KUKA KRL program: MyProgram_107().src

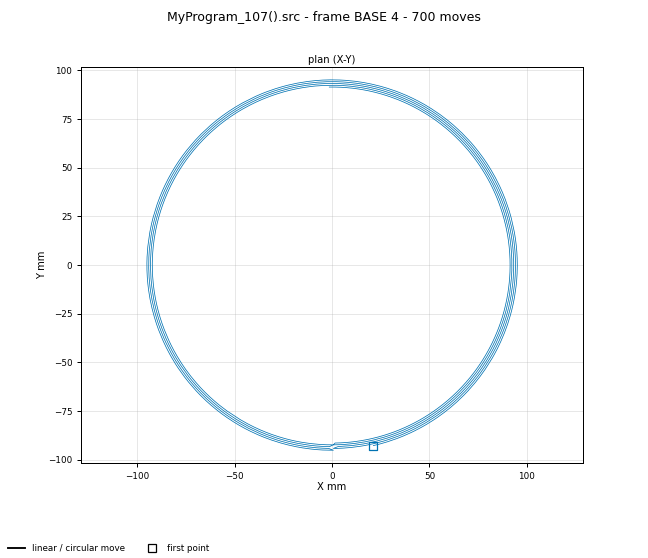
[picture p0: tool path of MyProgram_107().src in frame BASE 4, 700 of 700 moves have a stored position in this frame; points joined in program order, loops and branches not executed]
&ACCESS RVP
&REL 1
&PARAM TEMPLATE = C:\KRC\Roboter\Template\vorgabe
&PARAM EDITMASK = *
DEF MyProgram_107()
; ---- Setting reference (Base) ----
$BASE = BASE_DATA[4]

; --------------------------
; ---- Setting tool (TCP) ----
$TOOL = TOOL_DATA[3]
; --------------------------

$VEL.CP = VEL_APROX_PRINT
Startdeposition()
$VEL.CP = VEL_PRINT
LIN {X 21.2015,Y -92.7621,Z 95,A -81.1872,B 24.9355,C -1.8549,E1 25.0369,E2 526.4414} C_DIS
LIN {X 24.5046,Y -91.9451,Z 95,A -78.7968,B 24.9345,C -1.8695,E1 25.0434,E2 524.0201} C_DIS
LIN {X 28.303,Y -90.8473,Z 95,A -76.2009,B 24.9337,C -1.8802,E1 25.0504,E2 521.4036} C_DIS
LIN {X 33.1897,Y -89.179,Z 95,A -73.7268,B 24.9351,C -1.8608,E1 25.0568,E2 518.9806} C_DIS
LIN {X 36.3029,Y -87.9579,Z 95,A -71.0756,B 24.9332,C -1.8872,E1 25.0638,E2 516.2727} C_DIS
LIN {X 40.3024,Y -86.1975,Z 95,A -68.9078,B 24.9342,C -1.8741,E1 25.0692,E2 514.1415} C_DIS
LIN {X 42.5134,Y -85.1291,Z 95,A -67.3385,B 24.9338,C -1.8798,E1 25.0731,E2 512.5627} C_DIS
LIN {X 45.732,Y -83.4447,Z 95,A -64.735,B 24.9324,C -1.8992,E1 25.0796,E2 509.921} C_DIS
LIN {X 48.7101,Y -81.7418,Z 95,A -63.2036,B 24.9335,C -1.8829,E1 25.0832,E2 508.4327} C_DIS
LIN {X 51.7631,Y -79.8438,Z 95,A -61.164,B 24.9335,C -1.8824,E1 25.088,E2 506.4009} C_DIS
LIN {X 54.2431,Y -78.1791,Z 95,A -58.5386,B 24.9311,C -1.9172,E1 25.0942,E2 503.7022} C_DIS
LIN {X 57.6507,Y -75.7031,Z 95,A -56.3016,B 24.9315,C -1.9112,E1 25.0991,E2 501.4876} C_DIS
LIN {X 60.7617,Y -73.2277,Z 95,A -54.3783,B 24.9324,C -1.8987,E1 25.1032,E2 499.6011} C_DIS
LIN {X 64.0072,Y -70.4098,Z 95,A -51.4612,B 24.9311,C -1.9171,E1 25.1094,E2 496.6521} C_DIS
LIN {X 67.7886,Y -66.7757,Z 95,A -48.695,B 24.9316,C -1.9098,E1 25.1148,E2 493.9147} C_DIS
LIN {X 69.7218,Y -64.757,Z 95,A -46.6796,B 24.9304,C -1.9267,E1 25.1187,E2 491.8682} C_DIS
LIN {X 73.3658,Y -60.5954,Z 95,A -42.867,B 24.9284,C -1.9539,E1 25.1257,E2 488.0088} C_DIS
LIN {X 76.0575,Y -57.1798,Z 95,A -41.0314,B 24.9301,C -1.9308,E1 25.1287,E2 486.2364} C_DIS
LIN {X 78.597,Y -53.6362,Z 95,A -38.149,B 24.9289,C -1.9479,E1 25.1333,E2 483.3277} C_DIS
LIN {X 82.226,Y -47.8902,Z 95,A -34.4845,B 24.9292,C -1.9431,E1 25.1387,E2 479.6932} C_DIS
LIN {X 83.3859,Y -45.8405,Z 95,A -32.811,B 24.9282,C -1.9571,E1 25.141,E2 477.9955} C_DIS
LIN {X 84.9406,Y -42.8903,Z 95,A -31.1089,B 24.9286,C -1.9513,E1 25.1431,E2 476.3162} C_DIS
LIN {X 86.6182,Y -39.3911,Z 95,A -28.193,B 24.9264,C -1.9807,E1 25.1466,E2 473.3466} C_DIS
LIN {X 88.5125,Y -34.9259,Z 95,A -25.3594,B 24.926,C -1.9862,E1 25.1496,E2 470.5155} C_DIS
LIN {X 90.2327,Y -30.2054,Z 95,A -22.6628,B 24.9263,C -1.9829,E1 25.152,E2 467.8419} C_DIS
LIN {X 91.5044,Y -26.1004,Z 95,A -19.9815,B 24.9254,C -1.9946,E1 25.1542,E2 465.1482} C_DIS
LIN {X 92.2435,Y -23.3564,Z 95,A -18.4107,B 24.9254,C -1.9946,E1 25.1553,E2 463.5865} C_DIS
LIN {X 92.9574,Y -20.327,Z 95,A -16.5699,B 24.9251,C -1.9993,E1 25.1564,E2 461.7454} C_DIS
LIN {X 93.6612,Y -16.7881,Z 95,A -14.0181,B 24.9234,C -2.021,E1 25.1577,E2 459.1574} C_DIS
LIN {X 94.5474,Y -10.7315,Z 95,A -10.8838,B 24.9241,C -2.0114,E1 25.1589,E2 456.0642} C_DIS
LIN {X 94.8412,Y -7.7091,Z 95,A -9.0035,B 24.9235,C -2.0193,E1 25.1594,E2 454.1764} C_DIS
LIN {X 95.0524,Y -4.4048,Z 95,A -6.2816,B 24.9209,C -2.054,E1 25.1597,E2 451.3887} C_DIS
LIN {X 95.1533,Y -0.3254,Z 95,A -5.0589,B 24.9239,C -2.0141,E1 25.1598,E2 450.2674} C_DIS
LIN {X 95.0895,Y 3.5435,Z 95,A -2.1708,B 24.9217,C -2.043,E1 25.1596,E2 447.3283} C_DIS
LIN {X 94.9193,Y 6.6832,Z 95,A -0.2501,B 24.9212,C -2.0502,E1 25.1593,E2 445.4021} C_DIS
LIN {X 94.6098,Y 10.1644,Z 95,A 1.8084,B 24.9208,C -2.0551,E1 25.1587,E2 443.3443} C_DIS
LIN {X 94.2037,Y 13.414,Z 95,A 3.6958,B 24.9206,C -2.058,E1 25.158,E2 441.461} C_DIS
LIN {X 93.6507,Y 16.8467,Z 95,A 6.0545,B 24.9193,C -2.0748,E1 25.1569,E2 439.0765} C_DIS
LIN {X 92.0458,Y 24.1257,Z 95,A 10.1238,B 24.9195,C -2.0725,E1 25.1543,E2 435.0364} C_DIS
LIN {X 91.0638,Y 27.6036,Z 95,A 12.7765,B 24.9175,C -2.0973,E1 25.1522,E2 432.3402} C_DIS
LIN {X 88.9541,Y 33.7852,Z 95,A 16.3153,B 24.9178,C -2.0938,E1 25.1489,E2 428.8295} C_DIS
LIN {X 87.4635,Y 37.4746,Z 95,A 18.5781,B 24.9176,C -2.0957,E1 25.1465,E2 426.5748} C_DIS
LIN {X 86.1854,Y 40.3285,Z 95,A 20.5012,B 24.9171,C -2.1025,E1 25.1443,E2 424.6459} C_DIS
LIN {X 83.8275,Y 45.0262,Z 95,A 23.5493,B 24.9168,C -2.1068,E1 25.1404,E2 421.6038} C_DIS
LIN {X 81.6376,Y 48.8863,Z 95,A 26.2374,B 24.9161,C -2.1146,E1 25.1367,E2 418.9114} C_DIS
LIN {X 79.5978,Y 52.1396,Z 95,A 28.7064,B 24.9152,C -2.1265,E1 25.1329,E2 416.4267} C_DIS
LIN {X 77.8338,Y 54.7397,Z 95,A 30.587,B 24.9148,C -2.1308,E1 25.13,E2 414.5451} C_DIS
LIN {X 75.3135,Y 58.1563,Z 95,A 33.1694,B 24.9143,C -2.1381,E1 25.1256,E2 411.9578} C_DIS
LIN {X 72.7585,Y 61.3247,Z 95,A 35.3735,B 24.9145,C -2.1346,E1 25.1217,E2 409.7722} C_DIS
LIN {X 71.2409,Y 63.0815,Z 95,A 38.2884,B 24.9096,C -2.1951,E1 25.1161,E2 406.7272} C_DIS
LIN {X 66.7779,Y 67.7864,Z 95,A 42.0486,B 24.9094,C -2.1978,E1 25.1086,E2 402.9765} C_DIS
LIN {X 62.3108,Y 71.915,Z 95,A 44.542,B 24.9124,C -2.1611,E1 25.1036,E2 400.5797} C_DIS
LIN {X 59.3425,Y 74.3836,Z 95,A 46.9,B 24.9119,C -2.1667,E1 25.0985,E2 398.2176} C_DIS
LIN {X 55.6118,Y 77.2125,Z 95,A 49.4418,B 24.9124,C -2.1614,E1 25.0928,E2 395.6973} C_DIS
LIN {X 50.9589,Y 80.3585,Z 95,A 53.3712,B 24.9103,C -2.1869,E1 25.0836,E2 391.7206} C_DIS
LIN {X 47.6349,Y 82.3727,Z 95,A 55.2828,B 24.9113,C -2.1746,E1 25.079,E2 389.8439} C_DIS
LIN {X 44.3048,Y 84.2102,Z 95,A 57.5131,B 24.9113,C -2.1755,E1 25.0736,E2 387.6178} C_DIS
LIN {X 41.4825,Y 85.6362,Z 95,A 59.4743,B 24.9109,C -2.18,E1 25.0687,E2 385.6514} C_DIS
LIN {X 38.5041,Y 87.0171,Z 95,A 62.1318,B 24.9086,C -2.2069,E1 25.0617,E2 382.9366} C_DIS
LIN {X 34.8006,Y 88.5618,Z 95,A 63.6448,B 24.9111,C -2.1767,E1 25.058,E2 381.4986} C_DIS
LIN {X 32.3538,Y 89.485,Z 95,A 65.4865,B 24.9102,C -2.1877,E1 25.0531,E2 379.6347} C_DIS
LIN {X 28.4229,Y 90.8101,Z 95,A 68.3137,B 24.9091,C -2.2015,E1 25.0455,E2 376.78} C_DIS
LIN {X 24.6309,Y 91.9109,Z 95,A 70.369,B 24.9099,C -2.1916,E1 25.0401,E2 374.7517} C_DIS
LIN {X 20.202,Y 92.9847,Z 95,A 72.7708,B 24.9108,C -2.1809,E1 25.0336,E2 372.3785} C_DIS
LIN {X 16.1674,Y 93.7716,Z 95,A 75.332,B 24.9105,C -2.1849,E1 25.0266,E2 369.8107} C_DIS
LIN {X 11.8781,Y 94.4103,Z 95,A 78.3599,B 24.9092,C -2.2003,E1 25.0181,E2 366.7491} C_DIS
LIN {X 6.8428,Y 94.9085,Z 95,A 81.088,B 24.9101,C -2.1893,E1 25.0106,E2 364.0485} C_DIS
LIN {X 3.8615,Y 95.0758,Z 95,A 83.0082,B 24.9097,C -2.1935,E1 25.0052,E2 362.1189} C_DIS
LIN {X -0.7494,Y 95.1511,Z 95,A 85.9179,B 24.9094,C -2.1977,E1 24.9971,E2 359.1996} C_DIS
LIN {X -4.7837,Y 95.0348,Z 95,A 88.2592,B 24.9097,C -2.1938,E1 24.9906,E2 356.8671} C_DIS
LIN {X -8.378,Y 94.7851,Z 95,A 91.1031,B 24.9079,C -2.2161,E1 24.9825,E2 353.9688} C_DIS
LIN {X -12.6946,Y 94.3045,Z 95,A 92.7842,B 24.9107,C -2.1824,E1 24.9781,E2 352.3667} C_DIS
LIN {X -18.097,Y 93.4172,Z 95,A 96.3346,B 24.9102,C -2.1886,E1 24.9682,E2 348.7981} C_DIS
LIN {X -22.6473,Y 92.4196,Z 95,A 99.2215,B 24.9102,C -2.1888,E1 24.9604,E2 345.9069} C_DIS
LIN {X -25.4908,Y 91.6765,Z 95,A 101.4698,B 24.9089,C -2.2032,E1 24.9542,E2 343.6207} C_DIS
LIN {X -29.1325,Y 90.5847,Z 95,A 102.7942,B 24.9118,C -2.168,E1 24.9509,E2 342.3778} C_DIS
LIN {X -33.9169,Y 88.9043,Z 95,A 106.0614,B 24.9116,C -2.1712,E1 24.9423,E2 339.0964} C_DIS
LIN {X -36.0474,Y 88.0618,Z 95,A 107.6765,B 24.9111,C -2.1772,E1 24.9381,E2 337.4635} C_DIS
LIN {X -39.3326,Y 86.6446,Z 95,A 109.7691,B 24.9115,C -2.172,E1 24.9327,E2 335.3783} C_DIS
LIN {X -45.8745,Y 83.3674,Z 95,A 114.0483,B 24.9125,C -2.1605,E1 24.9221,E2 331.1149} C_DIS
LIN {X -49.5131,Y 81.2572,Z 95,A 117.3841,B 24.9107,C -2.1825,E1 24.914,E2 327.7164} C_DIS
LIN {X -52.9216,Y 79.0812,Z 95,A 119.0064,B 24.9132,C -2.1509,E1 24.9104,E2 326.1641} C_DIS
LIN {X -56.1766,Y 76.8015,Z 95,A 122.1635,B 24.9116,C -2.1713,E1 24.9031,E2 322.9476} C_DIS
LIN {X -59.1508,Y 74.5351,Z 95,A 124.6272,B 24.9114,C -2.1734,E1 24.8977,E2 320.4696} C_DIS
LIN {X -62.5657,Y 71.6924,Z 95,A 126.5051,B 24.914,C -2.1412,E1 24.8938,E2 318.661} C_DIS
LIN {X -67.2255,Y 67.3442,Z 95,A 131.1704,B 24.9126,C -2.1592,E1 24.8843,E2 313.9336} C_DIS
LIN {X -70.2591,Y 64.1715,Z 95,A 133.1273,B 24.9149,C -2.1302,E1 24.8807,E2 312.0372} C_DIS
LIN {X -74.5327,Y 59.1539,Z 95,A 137.5933,B 24.9144,C -2.136,E1 24.8727,E2 307.5368} C_DIS
LIN {X -76.7249,Y 56.2811,Z 95,A 139.2239,B 24.9163,C -2.1125,E1 24.8701,E2 305.9543} C_DIS
LIN {X -78.8114,Y 53.3202,Z 95,A 141.4933,B 24.9166,C -2.1093,E1 24.8665,E2 303.6813} C_DIS
LIN {X -80.6663,Y 50.4699,Z 95,A 143.4446,B 24.9173,C -2.1005,E1 24.8636,E2 301.7412} C_DIS
LIN {X -82.418,Y 47.556,Z 95,A 146.1137,B 24.9161,C -2.1146,E1 24.8598,E2 299.0245} C_DIS
LIN {X -84.1912,Y 44.3408,Z 95,A 148.3338,B 24.9166,C -2.1084,E1 24.8569,E2 296.8074} C_DIS
LIN {X -85.8378,Y 41.0629,Z 95,A 149.8509,B 24.9189,C -2.0797,E1 24.8551,E2 295.3506} C_DIS
LIN {X -87.0219,Y 38.493,Z 95,A 152.3254,B 24.9174,C -2.0992,E1 24.8522,E2 292.816} C_DIS
LIN {X -88.4862,Y 34.9931,Z 95,A 154.4167,B 24.9184,C -2.086,E1 24.8501,E2 290.7444} C_DIS
LIN {X -89.9166,Y 31.1356,Z 95,A 156.579,B 24.9198,C -2.0683,E1 24.8481,E2 288.6122} C_DIS
LIN {X -91.9922,Y 24.3233,Z 95,A 160.9692,B 24.9206,C -2.058,E1 24.8447,E2 284.221} C_DIS
LIN {X -92.7379,Y 21.3065,Z 95,A 163.485,B 24.9194,C -2.0727,E1 24.8431,E2 281.6555} C_DIS
LIN {X -93.629,Y 16.9675,Z 95,A 165.3634,B 24.922,C -2.039,E1 24.8421,E2 279.8464} C_DIS
LIN {X -94.6916,Y 9.3829,Z 95,A 169.8316,B 24.9235,C -2.0195,E1 24.8405,E2 275.398} C_DIS
LIN {X -95.0617,Y 4.1892,Z 95,A 173.6299,B 24.9227,C -2.0305,E1 24.8398,E2 271.5507} C_DIS
LIN {X -95.1501,Y 0.9439,Z 95,A 175.2093,B 24.9241,C -2.0122,E1 24.8398,E2 270.0053} C_DIS
LIN {X -95.1195,Y -2.5816,Z 95,A 177.8819,B 24.9233,C -2.023,E1 24.84,E2 267.2909} C_DIS
LIN {X -94.9474,Y -6.2682,Z 95,A -179.9881,B 24.924,C -2.013,E1 24.8403,E2 265.1721} C_DIS
LIN {X -94.6682,Y -9.6066,Z 95,A -178.4372,B 24.9256,C -1.9917,E1 24.8408,E2 263.6627} C_DIS
LIN {X -94.2789,Y -12.8847,Z 95,A -175.614,B 24.9241,C -2.0122,E1 24.8419,E2 260.7737} C_DIS
LIN {X -93.5576,Y -17.3616,Z 95,A -173.9302,B 24.9272,C -1.9701,E1 24.8426,E2 259.1803} C_DIS
LIN {X -92.5339,Y -22.1785,Z 95,A -170.9352,B 24.9278,C -1.9618,E1 24.8444,E2 256.1874} C_DIS
LIN {X -91.3174,Y -26.749,Z 95,A -168.1013,B 24.9285,C -1.9527,E1 24.8465,E2 253.3588} C_DIS
LIN {X -90.2356,Y -30.1967,Z 95,A -165.649,B 24.9283,C -1.955,E1 24.8486,E2 250.8869} C_DIS
LIN {X -89.1137,Y -33.3638,Z 95,A -162.3786,B 24.9258,C -1.9896,E1 24.8519,E2 247.5155} C_DIS
LIN {X -86.8377,Y -38.9041,Z 95,A -159.375,B 24.928,C -1.9596,E1 24.8552,E2 244.5671} C_DIS
LIN {X -85.2361,Y -42.2975,Z 95,A -157.1578,B 24.9286,C -1.9519,E1 24.8579,E2 242.3562} C_DIS
LIN {X -83.592,Y -45.4604,Z 95,A -156.0522,B 24.9314,C -1.9123,E1 24.8593,E2 241.3391} C_DIS
LIN {X -82.5088,Y -47.398,Z 95,A -154.2605,B 24.9306,C -1.9234,E1 24.8618,E2 239.5116} C_DIS
LIN {X -80.5549,Y -50.6484,Z 95,A -152.0371,B 24.9312,C -1.9155,E1 24.865,E2 237.2958} C_DIS
LIN {X -79.0451,Y -52.975,Z 95,A -149.9173,B 24.9305,C -1.9259,E1 24.8683,E2 235.1406} C_DIS
LIN {X -75.7376,Y -57.6056,Z 95,A -146.7407,B 24.9317,C -1.9092,E1 24.8735,E2 231.9883} C_DIS
LIN {X -73.7803,Y -60.0898,Z 95,A -144.6443,B 24.9315,C -1.9111,E1 24.8772,E2 229.8777} C_DIS
LIN {X -69.9548,Y -64.503,Z 95,A -141.4422,B 24.9328,C -1.8927,E1 24.8831,E2 226.7049} C_DIS
LIN {X -67.8056,Y -66.7584,Z 95,A -139.2653,B 24.9324,C -1.8987,E1 24.8874,E2 224.5045} C_DIS
LIN {X -64.794,Y -69.6871,Z 95,A -136.8336,B 24.933,C -1.8902,E1 24.8923,E2 222.083} C_DIS
LIN {X -62.2647,Y -71.9551,Z 95,A -134.6704,B 24.933,C -1.8902,E1 24.8968,E2 219.9113} C_DIS
LIN {X -58.8746,Y -74.7534,Z 95,A -132.3458,B 24.9341,C -1.8745,E1 24.9018,E2 217.6152} C_DIS
LIN {X -56.6915,Y -76.4243,Z 95,A -130.4441,B 24.9338,C -1.8798,E1 24.9061,E2 215.6941} C_DIS
LIN {X -53.9195,Y -78.404,Z 95,A -127.7984,B 24.9326,C -1.8966,E1 24.9123,E2 212.9995} C_DIS
LIN {X -50.599,Y -80.5857,Z 95,A -126.0845,B 24.9345,C -1.8699,E1 24.9162,E2 211.3436} C_DIS
LIN {X -47.9869,Y -82.1692,Z 95,A -123.7914,B 24.9336,C -1.8827,E1 24.9218,E2 209.0132} C_DIS
LIN {X -44.679,Y -84.0131,Z 95,A -121.931,B 24.9348,C -1.8653,E1 24.9263,E2 207.1888} C_DIS
LIN {X -41.8541,Y -85.4559,Z 95,A -119.2428,B 24.9331,C -1.8897,E1 24.9332,E2 204.4356} C_DIS
LIN {X -37.891,Y -87.2844,Z 95,A -117.5159,B 24.9354,C -1.8558,E1 24.9374,E2 202.7852} C_DIS
LIN {X -35.1955,Y -88.4067,Z 95,A -115.5498,B 24.9351,C -1.8612,E1 24.9425,E2 200.8019} C_DIS
LIN {X -31.1603,Y -89.9079,Z 95,A -112.6856,B 24.9346,C -1.8683,E1 24.9501,E2 197.915} C_DIS
LIN {X -26.3704,Y -91.4279,Z 95,A -109.6019,B 24.9346,C -1.8683,E1 24.9584,E2 194.8265} C_DIS
LIN {X -22.6878,Y -92.4097,Z 95,A -107.3277,B 24.9347,C -1.8662,E1 24.9646,E2 192.5538} C_DIS
LIN {X -18.4185,Y -93.3553,Z 95,A -105.0513,B 24.9357,C -1.8525,E1 24.9707,E2 190.3072} C_DIS
LIN {X -15.2065,Y -93.9323,Z 95,A -102.8454,B 24.9351,C -1.8604,E1 24.9768,E2 188.0804} C_DIS
LIN {X -10.5957,Y -94.5633,Z 95,A -100.3962,B 24.936,C -1.8474,E1 24.9835,E2 185.6603} C_DIS
LIN {X -8.0367,Y -94.815,Z 95,A -98.7449,B 24.9358,C -1.851,E1 24.9881,E2 183.9998} C_DIS
LIN {X -4.7799,Y -95.035,Z 95,A -96.5181,B 24.9351,C -1.8604,E1 24.9944,E2 181.7499} C_DIS
LIN {X 0.656,Y -95.1517,Z 95,A -93.9921,B 24.9369,C -1.8344,E1 25.0013,E2 179.2856} C_DIS
Enddeposition()
LIN {X 0.656,Y -95.1517,Z 95,A -93.9921,B 24.9369,C -1.8344,E1 25.0013,E2 179.2856} C_DIS
Startdeposition()
$VEL.CP = VEL_PRINT
LIN {X -1.8016,Y -94.2128,Z 95,A -96.3815,B 24.938,C -1.8192,E1 24.9945,E2 181.7111} C_DIS
LIN {X -5.0247,Y -94.0961,Z 95,A -97.8395,B 24.9368,C -1.8364,E1 24.9906,E2 183.1287} C_DIS
LIN {X -8.3046,Y -93.864,Z 95,A -99.7207,B 24.9365,C -1.8405,E1 24.9854,E2 185.001} C_DIS
LIN {X -12.2376,Y -93.4321,Z 95,A -102.7492,B 24.9379,C -1.8195,E1 24.9768,E2 188.0812} C_DIS
LIN {X -15.4201,Y -92.9598,Z 95,A -104.2663,B 24.9369,C -1.835,E1 24.9727,E2 189.5629} C_DIS
LIN {X -18.6733,Y -92.3617,Z 95,A -106.9067,B 24.9383,C -1.8145,E1 24.9654,E2 192.2549} C_DIS
LIN {X -22.444,Y -91.5182,Z 95,A -108.5274,B 24.9365,C -1.8403,E1 24.9611,E2 193.8166} C_DIS
LIN {X -26.32,Y -90.481,Z 95,A -111.1115,B 24.9367,C -1.837,E1 24.9541,E2 196.4127} C_DIS
LIN {X -28.7931,Y -89.7235,Z 95,A -113.5293,B 24.9386,C -1.81,E1 24.9476,E2 198.8989} C_DIS
LIN {X -33.2909,Y -88.1534,Z 95,A -115.5452,B 24.9364,C -1.8418,E1 24.9424,E2 200.8432} C_DIS
LIN {X -36.6065,Y -86.8289,Z 95,A -117.5659,B 24.9359,C -1.849,E1 24.9372,E2 202.8514} C_DIS
LIN {X -42.7686,Y -83.9652,Z 95,A -123.0072,B 24.9385,C -1.811,E1 24.9233,E2 208.3973} C_DIS
LIN {X -47.7528,Y -81.2344,Z 95,A -125.3815,B 24.9358,C -1.851,E1 24.9178,E2 210.6834} C_DIS
LIN {X -51.259,Y -79.0695,Z 95,A -128.4513,B 24.9368,C -1.8365,E1 24.9105,E2 213.7976} C_DIS
LIN {X -54.387,Y -76.9515,Z 95,A -130.1303,B 24.9351,C -1.8603,E1 24.9067,E2 215.4256} C_DIS
LIN {X -56.721,Y -75.2466,Z 95,A -131.7501,B 24.9346,C -1.8678,E1 24.9031,E2 217.0332} C_DIS
LIN {X -59.7224,Y -72.8888,Z 95,A -134.1379,B 24.9345,C -1.8698,E1 24.8979,E2 219.4251} C_DIS
LIN {X -62.4359,Y -70.5788,Z 95,A -136.5043,B 24.9346,C -1.8676,E1 24.8929,E2 221.8062} C_DIS
LIN {X -64.4138,Y -68.7764,Z 95,A -138.2964,B 24.9348,C -1.8656,E1 24.8892,E2 223.6103} C_DIS
LIN {X -67.4213,Y -65.8328,Z 95,A -140.7189,B 24.9341,C -1.8753,E1 24.8844,E2 226.0199} C_DIS
LIN {X -70.1048,Y -62.9654,Z 95,A -143.7724,B 24.9352,C -1.8596,E1 24.8786,E2 229.1245} C_DIS
LIN {X -72.9133,Y -59.6923,Z 95,A -145.7064,B 24.9332,C -1.8874,E1 24.8753,E2 231.0011} C_DIS
LIN {X -74.7444,Y -57.3812,Z 95,A -148.2796,B 24.9346,C -1.8671,E1 24.8708,E2 233.6348} C_DIS
LIN {X -77.4011,Y -53.7436,Z 95,A -150.2369,B 24.9324,C -1.8985,E1 24.8677,E2 235.527} C_DIS
LIN {X -79.1277,Y -51.1685,Z 95,A -152.1669,B 24.9322,C -1.9019,E1 24.8648,E2 237.4586} C_DIS
LIN {X -80.9682,Y -48.2031,Z 95,A -154.2751,B 24.9318,C -1.9079,E1 24.8617,E2 239.5633} C_DIS
LIN {X -82.859,Y -44.8742,Z 95,A -157.7343,B 24.9338,C -1.8791,E1 24.857,E2 243.1094} C_DIS
LIN {X -85.4064,Y -39.8127,Z 95,A -160.0394,B 24.9306,C -1.924,E1 24.8543,E2 245.3199} C_DIS
LIN {X -86.5711,Y -37.2147,Z 95,A -162.5817,B 24.9321,C -1.9038,E1 24.8515,E2 247.9245} C_DIS
LIN {X -88.1973,Y -33.1749,Z 95,A -164.5565,B 24.93,C -1.9323,E1 24.8495,E2 249.8424} C_DIS
LIN {X -89.4746,Y -29.5623,Z 95,A -166.7814,B 24.9293,C -1.9425,E1 24.8475,E2 252.0557} C_DIS
LIN {X -90.1989,Y -27.2709,Z 95,A -168.5198,B 24.9296,C -1.9383,E1 24.8461,E2 253.8141} C_DIS
LIN {X -91.3643,Y -23.0656,Z 95,A -171.0052,B 24.9286,C -1.9516,E1 24.8443,E2 256.2823} C_DIS
LIN {X -92.5133,Y -17.9053,Z 95,A -173.7797,B 24.9269,C -1.9752,E1 24.8427,E2 259.0168} C_DIS
LIN {X -93.1998,Y -13.8967,Z 95,A -176.8708,B 24.9277,C -1.9638,E1 24.8413,E2 262.1536} C_DIS
LIN {X -93.6028,Y -10.8545,Z 95,A -178.816,B 24.9274,C -1.9672,E1 24.8406,E2 264.1022} C_DIS
LIN {X -94.0154,Y -6.3559,Z 95,A 178.5563,B 24.9265,C -1.9796,E1 24.84,E2 266.7161} C_DIS
LIN {X -94.2181,Y -1.5135,Z 95,A 175.8516,B 24.9253,C -1.9965,E1 24.8398,E2 269.3967} C_DIS
LIN {X -94.1476,Y 3.9425,Z 95,A 171.7179,B 24.9263,C -1.9822,E1 24.8401,E2 273.5895} C_DIS
LIN {X -93.9007,Y 7.8801,Z 95,A 169.8809,B 24.9245,C -2.007,E1 24.8405,E2 275.3783} C_DIS
LIN {X -93.036,Y 14.9641,Z 95,A 165.7144,B 24.923,C -2.0262,E1 24.842,E2 279.5238} C_DIS
LIN {X -92.0758,Y 20.0337,Z 95,A 162.425,B 24.9226,C -2.0315,E1 24.8438,E2 282.8199} C_DIS
LIN {X -91.2971,Y 23.3269,Z 95,A 159.1952,B 24.9248,C -2.0024,E1 24.8461,E2 286.1382} C_DIS
LIN {X -89.7219,Y 28.7981,Z 95,A 156.9051,B 24.9213,C -2.0488,E1 24.8479,E2 288.3307} C_DIS
LIN {X -88.7648,Y 31.6277,Z 95,A 154.4671,B 24.9223,C -2.0354,E1 24.8502,E2 290.8146} C_DIS
LIN {X -87.477,Y 35.0336,Z 95,A 152.1408,B 24.9221,C -2.0387,E1 24.8526,E2 293.146} C_DIS
LIN {X -85.9536,Y 38.6171,Z 95,A 150.429,B 24.92,C -2.066,E1 24.8545,E2 294.8021} C_DIS
LIN {X -83.704,Y 43.2798,Z 95,A 146.7366,B 24.9205,C -2.0585,E1 24.8591,E2 298.5322} C_DIS
LIN {X -82.0732,Y 46.2974,Z 95,A 145.0703,B 24.9191,C -2.0775,E1 24.8613,E2 300.162} C_DIS
LIN {X -80.4047,Y 49.137,Z 95,A 143.146,B 24.9184,C -2.0856,E1 24.8641,E2 302.0768} C_DIS
LIN {X -78.3041,Y 52.4214,Z 95,A 140.6682,B 24.9182,C -2.0889,E1 24.8679,E2 304.5593} C_DIS
LIN {X -76.23,Y 55.3931,Z 95,A 138.7411,B 24.917,C -2.1035,E1 24.8709,E2 306.4609} C_DIS
LIN {X -74.0397,Y 58.2877,Z 95,A 135.763,B 24.9184,C -2.0854,E1 24.8761,E2 309.4962} C_DIS
LIN {X -71.7822,Y 61.046,Z 95,A 134.1277,B 24.9167,C -2.1076,E1 24.879,E2 311.0863} C_DIS
LIN {X -69.166,Y 63.9963,Z 95,A 131.2402,B 24.9174,C -2.0983,E1 24.8845,E2 314.0087} C_DIS
LIN {X -66.8819,Y 66.3789,Z 95,A 129.1146,B 24.9174,C -2.0994,E1 24.8887,E2 316.1406} C_DIS
LIN {X -64.1715,Y 69.0043,Z 95,A 127.3104,B 24.9157,C -2.1201,E1 24.8923,E2 317.9029} C_DIS
LIN {X -61.5187,Y 71.3795,Z 95,A 124.6603,B 24.9165,C -2.1098,E1 24.8979,E2 320.588} C_DIS
LIN {X -58.7598,Y 73.6665,Z 95,A 122.6428,B 24.9157,C -2.1196,E1 24.9023,E2 322.5898} C_DIS
LIN {X -54.9512,Y 76.5489,Z 95,A 120.1,B 24.9143,C -2.137,E1 24.9079,E2 325.1001} C_DIS
LIN {X -52.221,Y 78.4375,Z 95,A 118.3099,B 24.9134,C -2.1482,E1 24.912,E2 326.8694} C_DIS
LIN {X -47.4644,Y 81.4048,Z 95,A 114.5503,B 24.9138,C -2.1433,E1 24.921,E2 330.6525} C_DIS
LIN {X -45.0958,Y 82.7387,Z 95,A 112.86,B 24.9138,C -2.1449,E1 24.9251,E2 332.3437} C_DIS
LIN {X -39.0826,Y 85.7439,Z 95,A 108.865,B 24.913,C -2.1543,E1 24.9352,E2 336.3266} C_DIS
LIN {X -36.6824,Y 86.7969,Z 95,A 106.8857,B 24.9138,C -2.1442,E1 24.9403,E2 338.3347} C_DIS
LIN {X -31.6443,Y 88.759,Z 95,A 103.9098,B 24.9126,C -2.1586,E1 24.948,E2 341.2825} C_DIS
LIN {X -28.8431,Y 89.7073,Z 95,A 101.8686,B 24.9131,C -2.1528,E1 24.9535,E2 343.3412} C_DIS
LIN {X -24.4104,Y 91.0135,Z 95,A 98.5364,B 24.9142,C -2.1387,E1 24.9626,E2 346.712} C_DIS
LIN {X -19.8975,Y 92.1055,Z 95,A 96.0873,B 24.913,C -2.1534,E1 24.9691,E2 349.1292} C_DIS
LIN {X -16.6753,Y 92.7428,Z 95,A 94.0632,B 24.913,C -2.154,E1 24.9747,E2 351.1539} C_DIS
LIN {X -13.3371,Y 93.2814,Z 95,A 91.3766,B 24.9145,C -2.1347,E1 24.9823,E2 353.8885} C_DIS
LIN {X -7.7594,Y 93.9103,Z 95,A 89.0853,B 24.9114,C -2.1734,E1 24.9884,E2 356.089} C_DIS
LIN {X -2.7189,Y 94.1909,Z 95,A 86.1134,B 24.911,C -2.1778,E1 24.9967,E2 359.0513} C_DIS
LIN {X 2.2948,Y 94.2037,Z 95,A 82.9416,B 24.9113,C -2.1741,E1 25.0055,E2 362.2316} C_DIS
LIN {X 5.4769,Y 94.0711,Z 95,A 80.519,B 24.9127,C -2.1578,E1 25.0124,E2 364.6922} C_DIS
LIN {X 8.8708,Y 93.8118,Z 95,A 78.3952,B 24.9128,C -2.1557,E1 25.0183,E2 366.8195} C_DIS
LIN {X 12.4809,Y 93.4006,Z 95,A 76.6898,B 24.9115,C -2.1723,E1 25.0229,E2 368.4841} C_DIS
LIN {X 15.1025,Y 93.0129,Z 95,A 74.3812,B 24.9135,C -2.1481,E1 25.0295,E2 370.848} C_DIS
LIN {X 19.3197,Y 92.229,Z 95,A 72.7797,B 24.9107,C -2.1814,E1 25.0336,E2 372.3685} C_DIS
LIN {X 22.9943,Y 91.3826,Z 95,A 70.1813,B 24.9117,C -2.1695,E1 25.0407,E2 374.9913} C_DIS
LIN {X 25.7422,Y 90.6457,Z 95,A 67.611,B 24.9142,C -2.1394,E1 25.0478,E2 377.6287} C_DIS
LIN {X 30.3633,Y 89.2045,Z 95,A 65.4825,B 24.9121,C -2.1651,E1 25.0533,E2 379.6922} C_DIS
LIN {X 33.612,Y 88.0318,Z 95,A 63.6263,B 24.9115,C -2.1717,E1 25.0581,E2 381.5289} C_DIS
LIN {X 37.1817,Y 86.5852,Z 95,A 60.8602,B 24.9129,C -2.1544,E1 25.0653,E2 384.3297} C_DIS
LIN {X 40.8185,Y 84.9302,Z 95,A 58.3718,B 24.9133,C -2.1494,E1 25.0716,E2 386.8233} C_DIS
LIN {X 45.3869,Y 82.5808,Z 95,A 55.5484,B 24.9128,C -2.1558,E1 25.0785,E2 389.6235} C_DIS
LIN {X 47.7531,Y 81.2342,Z 95,A 53.2522,B 24.9148,C -2.1308,E1 25.0842,E2 391.9719} C_DIS
LIN {X 51.2882,Y 79.0508,Z 95,A 50.9509,B 24.9145,C -2.1348,E1 25.0895,E2 394.2563} C_DIS
LIN {X 54.0304,Y 77.2017,Z 95,A 49.6249,B 24.9128,C -2.1559,E1 25.0924,E2 395.5279} C_DIS
LIN {X 56.3155,Y 75.5512,Z 95,A 47.6529,B 24.9138,C -2.1436,E1 25.0969,E2 397.5218} C_DIS
LIN {X 59.905,Y 72.7383,Z 95,A 44.8788,B 24.9142,C -2.1385,E1 25.103,E2 400.2978} C_DIS
LIN {X 64.9917,Y 68.2325,Z 95,A 40.7583,B 24.9149,C -2.1306,E1 25.1115,E2 404.4203} C_DIS
LIN {X 66.8863,Y 66.3744,Z 95,A 38.2798,B 24.9176,C -2.096,E1 25.1165,E2 406.97} C_DIS
LIN {X 70.3455,Y 62.6965,Z 95,A 36.1252,B 24.9155,C -2.1221,E1 25.1204,E2 409.0533} C_DIS
LIN {X 72.0344,Y 60.7501,Z 95,A 34.3423,B 24.9165,C -2.1106,E1 25.1237,E2 410.8553} C_DIS
LIN {X 74.6839,Y 57.4597,Z 95,A 31.8086,B 24.9168,C -2.1057,E1 25.128,E2 413.3886} C_DIS
LIN {X 77.2662,Y 53.9377,Z 95,A 29.4476,B 24.9165,C -2.1099,E1 25.1319,E2 415.7283} C_DIS
LIN {X 79.2058,Y 51.0468,Z 95,A 27.3243,B 24.917,C -2.1042,E1 25.1351,E2 417.8544} C_DIS
LIN {X 80.9826,Y 48.1788,Z 95,A 24.8211,B 24.9187,C -2.0822,E1 25.1388,E2 420.3968} C_DIS
LIN {X 82.6256,Y 45.3043,Z 95,A 23.2106,B 24.918,C -2.0916,E1 25.1409,E2 421.9768} C_DIS
LIN {X 84.9204,Y 40.839,Z 95,A 20.2574,B 24.9183,C -2.0868,E1 25.1446,E2 424.9256} C_DIS
LIN {X 86.0432,Y 38.4184,Z 95,A 18.403,B 24.9194,C -2.0736,E1 25.1468,E2 426.8012} C_DIS
LIN {X 87.7631,Y 34.3069,Z 95,A 16.0388,B 24.919,C -2.0786,E1 25.1492,E2 429.1405} C_DIS
LIN {X 89.1848,Y 30.4218,Z 95,A 12.4457,B 24.9226,C -2.0312,E1 25.1526,E2 432.8251} C_DIS
LIN {X 90.7211,Y 25.4759,Z 95,A 10.3577,B 24.9203,C -2.061,E1 25.1542,E2 434.8308} C_DIS
LIN {X 92.2583,Y 19.1768,Z 95,A 6.3257,B 24.9215,C -2.0455,E1 25.1568,E2 438.8761} C_DIS
LIN {X 92.9454,Y 15.5066,Z 95,A 4.188,B 24.9217,C -2.0434,E1 25.1578,E2 441.0062} C_DIS
LIN {X 93.4353,Y 12.2127,Z 95,A 2.1245,B 24.9223,C -2.0356,E1 25.1586,E2 443.0761} C_DIS
LIN {X 93.8302,Y 8.6712,Z 95,A -0.0519,B 24.9229,C -2.0283,E1 25.1592,E2 445.2567} C_DIS
LIN {X 94.0832,Y 5.2588,Z 95,A -2.0806,B 24.9232,C -2.0236,E1 25.1596,E2 447.2844} C_DIS
LIN {X 94.2141,Y 1.7337,Z 95,A -4.211,B 24.9237,C -2.0173,E1 25.1598,E2 449.417} C_DIS
LIN {X 94.2218,Y -1.3039,Z 95,A -6.8075,B 24.9263,C -1.9833,E1 25.1597,E2 452.0784} C_DIS
LIN {X 94.0619,Y -5.6439,Z 95,A -8.6983,B 24.9248,C -2.0028,E1 25.1594,E2 453.9118} C_DIS
LIN {X 93.8245,Y -8.7333,Z 95,A -10.4345,B 24.9248,C -2.0024,E1 25.159,E2 455.6388} C_DIS
LIN {X 93.2035,Y -13.8809,Z 95,A -13.8781,B 24.9264,C -1.9812,E1 25.1578,E2 459.112} C_DIS
LIN {X 92.3936,Y -18.5181,Z 95,A -16.5445,B 24.9265,C -1.9794,E1 25.1564,E2 461.7669} C_DIS
LIN {X 91.7131,Y -21.6379,Z 95,A -18.3198,B 24.9265,C -1.9795,E1 25.1553,E2 463.5318} C_DIS
LIN {X 90.5738,Y -25.9958,Z 95,A -21.2367,B 24.9277,C -1.9642,E1 25.1532,E2 466.4682} C_DIS
LIN {X 89.4912,Y -29.511,Z 95,A -23.472,B 24.9282,C -1.9572,E1 25.1513,E2 468.7072} C_DIS
LIN {X 88.3537,Y -32.7594,Z 95,A -25.3223,B 24.928,C -1.9598,E1 25.1496,E2 470.5408} C_DIS
LIN {X 87.3502,Y -35.3451,Z 95,A -27.8318,B 24.9306,C -1.9239,E1 25.1469,E2 473.1214} C_DIS
LIN {X 85.7132,Y -39.1507,Z 95,A -29.7215,B 24.9295,C -1.9397,E1 25.1448,E2 474.9634} C_DIS
LIN {X 84.4593,Y -41.7843,Z 95,A -31.4628,B 24.9298,C -1.9357,E1 25.1426,E2 476.705} C_DIS
LIN {X 82.75,Y -45.0751,Z 95,A -33.7029,B 24.9302,C -1.9296,E1 25.1397,E2 478.9476} C_DIS
LIN {X 81.2821,Y -47.672,Z 95,A -35.8803,B 24.9316,C -1.9108,E1 25.1366,E2 481.1582} C_DIS
LIN {X 78.2798,Y -52.4542,Z 95,A -39.3344,B 24.9323,C -1.9004,E1 25.1313,E2 484.6196} C_DIS
LIN {X 76.3215,Y -55.2682,Z 95,A -40.7563,B 24.9309,C -1.9192,E1 25.1291,E2 485.99} C_DIS
LIN {X 74.9196,Y -57.1524,Z 95,A -42.8885,B 24.9331,C -1.8893,E1 25.1254,E2 488.1828} C_DIS
LIN {X 72.7051,Y -59.945,Z 95,A -44.5977,B 24.9323,C -1.9005,E1 25.1224,E2 489.8577} C_DIS
LIN {X 69.9525,Y -63.1355,Z 95,A -47.1184,B 24.9326,C -1.8954,E1 25.1178,E2 492.3789} C_DIS
LIN {X 68.0962,Y -65.1332,Z 95,A -49.3716,B 24.9345,C -1.8694,E1 25.1133,E2 494.6839} C_DIS
LIN {X 65.2837,Y -67.9512,Z 95,A -51.1708,B 24.9333,C -1.8864,E1 25.1098,E2 496.4354} C_DIS
LIN {X 62.3776,Y -70.6289,Z 95,A -53.6092,B 24.9338,C -1.8795,E1 25.1047,E2 498.8802} C_DIS
LIN {X 60.2802,Y -72.4265,Z 95,A -55.8704,B 24.9355,C -1.8545,E1 25.0998,E2 501.1919} C_DIS
LIN {X 57.0154,Y -75.0255,Z 95,A -58.3975,B 24.9359,C -1.8495,E1 25.0941,E2 503.7217} C_DIS
LIN {X 53.7411,Y -77.4028,Z 95,A -60.1101,B 24.9343,C -1.8717,E1 25.0904,E2 505.3759} C_DIS
LIN {X 48.5269,Y -80.7754,Z 95,A -64.2239,B 24.9357,C -1.8522,E1 25.0806,E2 509.5226} C_DIS
LIN {X 44.9637,Y -82.8104,Z 95,A -66.4102,B 24.9352,C -1.859,E1 25.0753,E2 511.6864} C_DIS
LIN {X 42.0537,Y -84.3258,Z 95,A -68.212,B 24.935,C -1.8626,E1 25.0709,E2 513.4746} C_DIS
LIN {X 39.8398,Y -85.3937,Z 95,A -70.5867,B 24.9373,C -1.8286,E1 25.0647,E2 515.9237} C_DIS
LIN {X 35.9744,Y -87.0941,Z 95,A -72.4519,B 24.9358,C -1.85,E1 25.06,E2 517.7339} C_DIS
LIN {X 33.6408,Y -88.0209,Z 95,A -74.2614,B 24.9367,C -1.8378,E1 25.0552,E2 519.5684} C_DIS
LIN {X 29.2694,Y -89.5694,Z 95,A -76.7848,B 24.9362,C -1.8448,E1 25.0486,E2 522.0702} C_DIS
LIN {X 26.5305,Y -90.4185,Z 95,A -79.3966,B 24.9384,C -1.8121,E1 25.0414,E2 524.7549} C_DIS
LIN {X 21.8649,Y -91.6595,Z 95,A -82.2936,B 24.9386,C -1.8106,E1 25.0335,E2 527.6513} C_DIS
LIN {X 17.2725,Y -92.6351,Z 95,A -84.3172,B 24.9367,C -1.8374,E1 25.0282,E2 529.6092} C_DIS
LIN {X 14.5797,Y -93.0955,Z 95,A -86.1319,B 24.9372,C -1.8307,E1 25.0231,E2 531.4378} C_DIS
LIN {X 9.9086,Y -93.7077,Z 95,A -89.5656,B 24.9386,C -1.8093,E1 25.0135,E2 534.92} C_DIS
LIN {X 5.5629,Y -94.0664,Z 95,A -91.4621,B 24.9369,C -1.8342,E1 25.0084,E2 536.7564} C_DIS
LIN {X 2.5065,Y -94.1975,Z 95,A -93.1285,B 24.9365,C -1.8404,E1 25.0038,E2 538.4079} C_DIS
LIN {X 0.6564,Y -94.2138,Z 95,A -94.3706,B 24.9368,C -1.8362,E1 25.0003,E2 539.6596} C_DIS
Enddeposition()
LIN {X 0.6564,Y -94.2138,Z 95,A -94.3706,B 24.9368,C -1.8362,E1 25.0003,E2 539.6596} C_DIS
Startdeposition()
$VEL.CP = VEL_PRINT
LIN {X 3.1308,Y -93.254,Z 95,A -92.0019,B 24.9336,C -1.8821,E1 25.0072,E2 537.1824} C_DIS
LIN {X 10.2868,Y -92.7391,Z 95,A -87.7242,B 24.9338,C -1.8797,E1 25.0191,E2 532.9127} C_DIS
LIN {X 15.9545,Y -91.9337,Z 95,A -84.2582,B 24.9338,C -1.8804,E1 25.0286,E2 529.4483} C_DIS
LIN {X 19.0057,Y -91.3501,Z 95,A -81.9048,B 24.9325,C -1.8979,E1 25.0352,E2 527.0561} C_DIS
LIN {X 23.2348,Y -90.3669,Z 95,A -79.1226,B 24.932,C -1.9048,E1 25.0427,E2 524.2619} C_DIS
LIN {X 28.4266,Y -88.871,Z 95,A -76.2617,B 24.9329,C -1.8921,E1 25.0503,E2 521.4361} C_DIS
LIN {X 31.4975,Y -87.8305,Z 95,A -73.9088,B 24.9318,C -1.9077,E1 25.0566,E2 519.051} C_DIS
LIN {X 35.6459,Y -86.2303,Z 95,A -71.1083,B 24.9313,C -1.9142,E1 25.0638,E2 516.2417} C_DIS
LIN {X 39.0703,Y -84.7329,Z 95,A -69.2111,B 24.9321,C -1.9032,E1 25.0686,E2 514.3752} C_DIS
LIN {X 42.1742,Y -83.2315,Z 95,A -67.1619,B 24.9321,C -1.9042,E1 25.0737,E2 512.3292} C_DIS
LIN {X 45.0007,Y -81.739,Z 95,A -65.0643,B 24.9314,C -1.9125,E1 25.0789,E2 510.2179} C_DIS
LIN {X 48.3432,Y -79.8059,Z 95,A -62.4451,B 24.9305,C -1.926,E1 25.0852,E2 507.5748} C_DIS
LIN {X 51.5083,Y -77.8008,Z 95,A -60.4753,B 24.931,C -1.9182,E1 25.0898,E2 505.6298} C_DIS
LIN {X 54.3519,Y -75.8415,Z 95,A -58.2646,B 24.9305,C -1.9259,E1 25.0949,E2 503.4086} C_DIS
LIN {X 56.8955,Y -73.9523,Z 95,A -55.9359,B 24.9291,C -1.9443,E1 25.1001,E2 501.0451} C_DIS
LIN {X 59.6811,Y -71.7231,Z 95,A -54.442,B 24.9307,C -1.9232,E1 25.1032,E2 499.6065} C_DIS
LIN {X 62.9064,Y -68.9121,Z 95,A -51.4689,B 24.9293,C -1.9421,E1 25.1095,E2 496.6007} C_DIS
LIN {X 66.4056,Y -65.5464,Z 95,A -48.3885,B 24.9285,C -1.953,E1 25.1156,E2 493.5074} C_DIS
LIN {X 68.9851,Y -62.8268,Z 95,A -46.0832,B 24.9281,C -1.959,E1 25.12,E2 491.1983} C_DIS
LIN {X 72.4359,Y -58.814,Z 95,A -42.5494,B 24.9266,C -1.9782,E1 25.1263,E2 487.6354} C_DIS
LIN {X 74.8895,Y -55.6582,Z 95,A -40.6815,B 24.9278,C -1.9627,E1 25.1294,E2 485.8131} C_DIS
LIN {X 76.9462,Y -52.779,Z 95,A -37.8635,B 24.9255,C -1.9931,E1 25.1339,E2 482.9371} C_DIS
LIN {X 79.2314,Y -49.2793,Z 95,A -35.9033,B 24.9267,C -1.9774,E1 25.1368,E2 481.0238} C_DIS
LIN {X 80.7166,Y -46.8081,Z 95,A -34.2007,B 24.9265,C -1.9799,E1 25.1392,E2 479.324} C_DIS
LIN {X 82.5161,Y -43.5561,Z 95,A -32.0837,B 24.9265,C -1.9804,E1 25.142,E2 477.217} C_DIS
LIN {X 84.0016,Y -40.6179,Z 95,A -29.9725,B 24.9258,C -1.9898,E1 25.1446,E2 475.0949} C_DIS
LIN {X 86.518,Y -34.9391,Z 95,A -26.1642,B 24.9249,C -2.0011,E1 25.1488,E2 471.2807} C_DIS
LIN {X 87.8621,Y -31.41,Z 95,A -23.7874,B 24.9242,C -2.0105,E1 25.1511,E2 468.8952} C_DIS
LIN {X 89.0593,Y -27.8303,Z 95,A -21.6507,B 24.9242,C -2.0109,E1 25.1529,E2 466.7696} C_DIS
LIN {X 90.0245,Y -24.5287,Z 95,A -19.6316,B 24.9239,C -2.014,E1 25.1545,E2 464.7547} C_DIS
LIN {X 90.7508,Y -21.6913,Z 95,A -17.9379,B 24.9239,C -2.0157,E1 25.1556,E2 463.0668} C_DIS
LIN {X 92.0207,Y -15.4347,Z 95,A -13.9149,B 24.9226,C -2.0321,E1 25.1578,E2 459.0286} C_DIS
LIN {X 92.8511,Y -9.2172,Z 95,A -10.1727,B 24.9219,C -2.0402,E1 25.1591,E2 455.2893} C_DIS
LIN {X 93.0614,Y -6.77,Z 95,A -8.1185,B 24.92,C -2.0658,E1 25.1595,E2 453.1868} C_DIS
LIN {X 93.2926,Y -1.5944,Z 95,A -5.2511,B 24.9201,C -2.0641,E1 25.1598,E2 450.3405} C_DIS
LIN {X 93.289,Y 1.7886,Z 95,A -3.2735,B 24.9199,C -2.067,E1 25.1598,E2 448.3678} C_DIS
LIN {X 93.1532,Y 5.3432,Z 95,A -1.0523,B 24.9192,C -2.0754,E1 25.1594,E2 446.14} C_DIS
LIN {X 92.8933,Y 8.7693,Z 95,A 0.9497,B 24.919,C -2.078,E1 25.1589,E2 444.1437} C_DIS
LIN {X 92.5349,Y 11.9721,Z 95,A 2.9468,B 24.9185,C -2.085,E1 25.1583,E2 442.142} C_DIS
LIN {X 92.0032,Y 15.5396,Z 95,A 5.382,B 24.9173,C -2.1003,E1 25.1572,E2 439.6851} C_DIS
LIN {X 91.3848,Y 18.8376,Z 95,A 7.4103,B 24.9169,C -2.1054,E1 25.1561,E2 437.6564} C_DIS
LIN {X 90.207,Y 23.8535,Z 95,A 10.3628,B 24.9167,C -2.1071,E1 25.1541,E2 434.717} C_DIS
LIN {X 89.2775,Y 27.1266,Z 95,A 12.9669,B 24.9147,C -2.1329,E1 25.152,E2 432.0669} C_DIS
LIN {X 88.1638,Y 30.55,Z 95,A 14.6637,B 24.9157,C -2.1201,E1 25.1505,E2 430.41} C_DIS
LIN {X 86.9994,Y 33.7242,Z 95,A 16.661,B 24.9155,C -2.1232,E1 25.1485,E2 428.4164} C_DIS
LIN {X 85.8582,Y 36.5309,Z 95,A 19.0175,B 24.9135,C -2.1472,E1 25.1459,E2 426.0162} C_DIS
LIN {X 84.4551,Y 39.6671,Z 95,A 20.6825,B 24.9144,C -2.1364,E1 25.144,E2 424.3855} C_DIS
LIN {X 81.4324,Y 45.55,Z 95,A 24.8092,B 24.9133,C -2.15,E1 25.1386,E2 420.2487} C_DIS
LIN {X 79.6819,Y 48.5473,Z 95,A 26.7663,B 24.9133,C -2.1491,E1 25.1358,E2 418.3036} C_DIS
LIN {X 77.6881,Y 51.6792,Z 95,A 29.0602,B 24.9129,C -2.1555,E1 25.1323,E2 416.0061} C_DIS
LIN {X 75.7889,Y 54.4257,Z 95,A 31.2115,B 24.9121,C -2.1644,E1 25.1288,E2 413.8443} C_DIS
LIN {X 73.7654,Y 57.138,Z 95,A 33.2003,B 24.912,C -2.1661,E1 25.1254,E2 411.8607} C_DIS
LIN {X 71.3103,Y 60.1754,Z 95,A 35.4677,B 24.912,C -2.167,E1 25.1214,E2 409.6019} C_DIS
LIN {X 69.3807,Y 62.389,Z 95,A 37.8222,B 24.9099,C -2.1913,E1 25.117,E2 407.2003} C_DIS
LIN {X 67.0483,Y 64.8891,Z 95,A 39.4531,B 24.911,C -2.1787,E1 25.1139,E2 405.6064} C_DIS
LIN {X 64.5128,Y 67.411,Z 95,A 41.6691,B 24.9105,C -2.184,E1 25.1094,E2 403.3871} C_DIS
LIN {X 60.6004,Y 70.9481,Z 95,A 44.8046,B 24.9103,C -2.1866,E1 25.1029,E2 400.2578} C_DIS
LIN {X 57.4914,Y 73.4914,Z 95,A 47.3312,B 24.9098,C -2.1934,E1 25.0974,E2 397.7248} C_DIS
LIN {X 54.6389,Y 75.6368,Z 95,A 49.4909,B 24.9095,C -2.196,E1 25.0925,E2 395.5665} C_DIS
LIN {X 51.6222,Y 77.7248,Z 95,A 52.7118,B 24.9063,C -2.2348,E1 25.0849,E2 392.2646} C_DIS
LIN {X 47.187,Y 80.4956,Z 95,A 54.8903,B 24.909,C -2.2022,E1 25.0798,E2 390.17} C_DIS
LIN {X 44.2005,Y 82.1733,Z 95,A 57.0802,B 24.9085,C -2.2081,E1 25.0745,E2 387.9723} C_DIS
LIN {X 39.9825,Y 84.3069,Z 95,A 59.8468,B 24.9086,C -2.2069,E1 25.0676,E2 385.216} C_DIS
LIN {X 34.3799,Y 86.7418,Z 95,A 63.3387,B 24.9091,C -2.2018,E1 25.0587,E2 381.7446} C_DIS
LIN {X 30.8294,Y 88.0658,Z 95,A 65.9013,B 24.9082,C -2.2122,E1 25.0519,E2 379.1627} C_DIS
LIN {X 26.0081,Y 89.6098,Z 95,A 68.9241,B 24.9082,C -2.2115,E1 25.0438,E2 376.147} C_DIS
LIN {X 23.463,Y 90.3083,Z 95,A 70.7028,B 24.9077,C -2.2181,E1 25.039,E2 374.3555} C_DIS
LIN {X 19.058,Y 91.3396,Z 95,A 73.1665,B 24.9085,C -2.2086,E1 25.0324,E2 371.9177} C_DIS
LIN {X 16.6029,Y 91.8171,Z 95,A 75.267,B 24.9068,C -2.2287,E1 25.0265,E2 369.7718} C_DIS
LIN {X 12.8029,Y 92.4242,Z 95,A 77.5994,B 24.9068,C -2.2283,E1 25.02,E2 367.4426} C_DIS
LIN {X 8.3881,Y 92.9285,Z 95,A 80.847,B 24.9053,C -2.2465,E1 25.0109,E2 364.1536} C_DIS
LIN {X 4.0833,Y 93.2168,Z 95,A 82.6941,B 24.9076,C -2.2189,E1 25.0059,E2 362.3727} C_DIS
LIN {X -2.0651,Y 93.2839,Z 95,A 86.1354,B 24.9086,C -2.2068,E1 24.9964,E2 358.9604} C_DIS
LIN {X -5.3094,Y 93.1551,Z 95,A 88.6198,B 24.9073,C -2.2227,E1 24.9894,E2 356.4377} C_DIS
LIN {X -8.1675,Y 92.9489,Z 95,A 91.3791,B 24.9045,C -2.2558,E1 24.9815,E2 353.5984} C_DIS
LIN {X -13.6972,Y 92.297,Z 95,A 93.5507,B 24.9083,C -2.2114,E1 24.9758,E2 351.5305} C_DIS
LIN {X -19.2168,Y 91.307,Z 95,A 96.9929,B 24.9085,C -2.2087,E1 24.9663,E2 348.0912} C_DIS
LIN {X -21.9943,Y 90.6769,Z 95,A 99.0507,B 24.9078,C -2.2173,E1 24.9607,E2 346.0101} C_DIS
LIN {X -26.7158,Y 89.3999,Z 95,A 101.9893,B 24.9082,C -2.212,E1 24.9528,E2 343.0795} C_DIS
LIN {X -30.3261,Y 88.242,Z 95,A 104.3445,B 24.9084,C -2.21,E1 24.9465,E2 340.7246} C_DIS
LIN {X -33.5888,Y 87.0526,Z 95,A 107.1061,B 24.9069,C -2.2279,E1 24.9392,E2 337.9145} C_DIS
LIN {X -37.3899,Y 85.4871,Z 95,A 108.8107,B 24.9094,C -2.1974,E1 24.935,E2 336.2786} C_DIS
LIN {X -41.2638,Y 83.6862,Z 95,A 111.7947,B 24.9088,C -2.205,E1 24.9274,E2 333.2688} C_DIS
LIN {X -45.801,Y 81.2923,Z 95,A 114.6552,B 24.91,C -2.1903,E1 24.9205,E2 330.4353} C_DIS
LIN {X -50.0214,Y 78.7661,Z 95,A 117.6259,B 24.9106,C -2.1831,E1 24.9134,E2 327.4725} C_DIS
LIN {X -52.2549,Y 77.3011,Z 95,A 119.3318,B 24.9106,C -2.1821,E1 24.9094,E2 325.7635} C_DIS
LIN {X -54.9722,Y 75.3932,Z 95,A 121.4609,B 24.9108,C -2.1808,E1 24.9046,E2 323.6299} C_DIS
LIN {X -58.3684,Y 72.797,Z 95,A 124.2305,B 24.9108,C -2.1798,E1 24.8985,E2 320.8525} C_DIS
LIN {X -60.7388,Y 70.8302,Z 95,A 126.0127,B 24.9115,C -2.1721,E1 24.8947,E2 319.0817} C_DIS
LIN {X -63.2718,Y 68.5768,Z 95,A 128.1474,B 24.9118,C -2.169,E1 24.8903,E2 316.9458} C_DIS
LIN {X -66.5379,Y 65.4124,Z 95,A 131.0408,B 24.912,C -2.1655,E1 24.8846,E2 314.0486} C_DIS
LIN {X -68.5252,Y 63.3281,Z 95,A 132.6792,B 24.9127,C -2.157,E1 24.8815,E2 312.4232} C_DIS
LIN {X -70.8791,Y 60.6814,Z 95,A 134.8434,B 24.9132,C -2.1512,E1 24.8775,E2 310.2633} C_DIS
LIN {X -73.5467,Y 57.4215,Z 95,A 137.6248,B 24.9132,C -2.1505,E1 24.8726,E2 307.4706} C_DIS
LIN {X -75.9916,Y 54.1416,Z 95,A 139.9935,B 24.9142,C -2.1392,E1 24.8687,E2 305.1173} C_DIS
LIN {X -77.888,Y 51.3759,Z 95,A 142.0727,B 24.9146,C -2.1341,E1 24.8655,E2 303.0398} C_DIS
LIN {X -79.6893,Y 48.5351,Z 95,A 144.128,B 24.9151,C -2.1279,E1 24.8625,E2 300.9888} C_DIS
LIN {X -82.3058,Y 43.9554,Z 95,A 147.537,B 24.9154,C -2.1238,E1 24.8579,E2 297.5717} C_DIS
LIN {X -83.8675,Y 40.8971,Z 95,A 149.5867,B 24.916,C -2.1157,E1 24.8553,E2 295.5302} C_DIS
LIN {X -85.325,Y 37.7617,Z 95,A 151.7275,B 24.9165,C -2.1099,E1 24.8529,E2 293.3916} C_DIS
LIN {X -87.922,Y 31.2393,Z 95,A 155.9208,B 24.9178,C -2.093,E1 24.8487,E2 289.2151} C_DIS
LIN {X -88.8776,Y 28.4063,Z 95,A 158.5002,B 24.9165,C -2.1105,E1 24.8464,E2 286.5793} C_DIS
LIN {X -90.0067,Y 24.5947,Z 95,A 159.9734,B 24.9194,C -2.0727,E1 24.8454,E2 285.1877} C_DIS
LIN {X -90.9746,Y 20.7301,Z 95,A 162.8101,B 24.9191,C -2.077,E1 24.8434,E2 282.324} C_DIS
LIN {X -91.9244,Y 16.006,Z 95,A 165.7713,B 24.9198,C -2.0676,E1 24.8419,E2 279.3677} C_DIS
LIN {X -92.6635,Y 10.9324,Z 95,A 168.8278,B 24.9208,C -2.0547,E1 24.8408,E2 276.3238} C_DIS
LIN {X -92.9817,Y 7.7823,Z 95,A 170.8909,B 24.921,C -2.0521,E1 24.8402,E2 274.2546} C_DIS
LIN {X -93.2468,Y 3.3639,Z 95,A 174.2797,B 24.9201,C -2.0643,E1 24.8398,E2 270.8163} C_DIS
LIN {X -93.3042,Y -0.5909,Z 95,A 176.0209,B 24.9223,C -2.0351,E1 24.8398,E2 269.1343} C_DIS
LIN {X -93.0615,Y -6.7689,Z 95,A -179.315,B 24.9212,C -2.05,E1 24.8405,E2 264.4065} C_DIS
LIN {X -92.6294,Y -11.2237,Z 95,A -177.5159,B 24.9241,C -2.0116,E1 24.8411,E2 262.6882} C_DIS
LIN {X -91.6986,Y -17.2502,Z 95,A -173.8337,B 24.9252,C -1.9979,E1 24.8427,E2 259.0168} C_DIS
LIN {X -91.0114,Y -20.5708,Z 95,A -171.7118,B 24.9255,C -1.9927,E1 24.8439,E2 256.8949} C_DIS
LIN {X -90.3555,Y -23.2791,Z 95,A -169.7697,B 24.9254,C -1.9947,E1 24.8452,E2 254.9367} C_DIS
LIN {X -89.3066,Y -27.0303,Z 95,A -167.5141,B 24.9263,C -1.9832,E1 24.847,E2 252.6956} C_DIS
LIN {X -88.5123,Y -29.5245,Z 95,A -165.7205,B 24.9262,C -1.9842,E1 24.8486,E2 250.8892} C_DIS
LIN {X -87.2809,Y -32.986,Z 95,A -163.2357,B 24.9262,C -1.9848,E1 24.851,E2 248.389} C_DIS
LIN {X -85.2839,Y -37.8546,Z 95,A -160.1753,B 24.9272,C -1.9701,E1 24.8543,E2 245.3467} C_DIS
LIN {X -83.9285,Y -40.7701,Z 95,A -157.5691,B 24.9261,C -1.9846,E1 24.8575,E2 242.6917} C_DIS
LIN {X -82.1259,Y -44.288,Z 95,A -155.8446,B 24.9283,C -1.9557,E1 24.8597,E2 241.0271} C_DIS
LIN {X -80.5102,Y -47.1622,Z 95,A -153.6929,B 24.9283,C -1.9543,E1 24.8627,E2 238.8675} C_DIS
LIN {X -77.9341,Y -51.3061,Z 95,A -150.8622,B 24.9293,C -1.9413,E1 24.8669,E2 236.0535} C_DIS
LIN {X -73.7509,Y -57.1568,Z 95,A -146.4892,B 24.9302,C -1.9289,E1 24.8741,E2 231.6888} C_DIS
LIN {X -72.2478,Y -59.046,Z 95,A -144.3879,B 24.9291,C -1.9453,E1 24.8779,E2 229.5387} C_DIS
LIN {X -69.6556,Y -62.082,Z 95,A -142.3362,B 24.9304,C -1.9268,E1 24.8816,E2 227.5217} C_DIS
LIN {X -67.2527,Y -64.677,Z 95,A -140.1703,B 24.9308,C -1.9219,E1 24.8857,E2 225.358} C_DIS
LIN {X -64.6818,Y -67.2481,Z 95,A -137.787,B 24.9308,C -1.9221,E1 24.8905,E2 222.9642} C_DIS
LIN {X -61.776,Y -69.9288,Z 95,A -135.3637,B 24.9311,C -1.9171,E1 24.8955,E2 220.5432} C_DIS
LIN {X -58.8683,Y -72.3918,Z 95,A -132.6295,B 24.9305,C -1.9257,E1 24.9015,E2 217.778} C_DIS
LIN {X -56.178,Y -74.499,Z 95,A -131.1566,B 24.9322,C -1.9014,E1 24.9046,E2 216.3576} C_DIS
LIN {X -53.4539,Y -76.4768,Z 95,A -128.0029,B 24.9299,C -1.934,E1 24.912,E2 213.1157} C_DIS
LIN {X -49.2899,Y -79.2248,Z 95,A -125.9798,B 24.9327,C -1.8947,E1 24.9166,E2 211.1797} C_DIS
LIN {X -46.746,Y -80.7523,Z 95,A -123.3681,B 24.931,C -1.9184,E1 24.9231,E2 208.5038} C_DIS
LIN {X -43.2045,Y -82.7013,Z 95,A -121.7797,B 24.9334,C -1.8853,E1 24.9268,E2 206.9897} C_DIS
LIN {X -40.972,Y -83.8308,Z 95,A -119.2788,B 24.9312,C -1.9157,E1 24.9333,E2 204.4099} C_DIS
LIN {X -37.1676,Y -85.584,Z 95,A -117.3763,B 24.933,C -1.8903,E1 24.938,E2 202.5632} C_DIS
LIN {X -33.96,Y -86.9067,Z 95,A -115.3082,B 24.9333,C -1.8861,E1 24.9433,E2 200.5005} C_DIS
LIN {X -29.1093,Y -88.6501,Z 95,A -112.3122,B 24.9339,C -1.8777,E1 24.9512,E2 197.5187} C_DIS
LIN {X -26.4366,Y -89.4827,Z 95,A -110.4363,B 24.9336,C -1.8818,E1 24.9562,E2 195.6298} C_DIS
LIN {X -22.0609,Y -90.6606,Z 95,A -107.7571,B 24.934,C -1.8767,E1 24.9635,E2 192.9589} C_DIS
LIN {X -17.6127,Y -91.6287,Z 95,A -105.3112,B 24.9349,C -1.8635,E1 24.9701,E2 190.5413} C_DIS
LIN {X -11.7531,Y -92.5633,Z 95,A -100.6249,B 24.9324,C -1.8984,E1 24.9832,E2 185.7681} C_DIS
LIN {X -8.1281,Y -92.9525,Z 95,A -99.0942,B 24.9342,C -1.8737,E1 24.9873,E2 184.2954} C_DIS
LIN {X -5.2694,Y -93.1573,Z 95,A -96.5451,B 24.9322,C -1.9013,E1 24.9946,E2 181.6799} C_DIS
LIN {X -1.3491,Y -93.2971,Z 95,A -93.9664,B 24.9318,C -1.9077,E1 25.0019,E2 179.0858} C_DIS
LIN {X -1.3491,Y -93.2971,Z 95,A -93.9664,B 24.9318,C -1.9077,E1 25.0019,E2 179.0858} C_DIS
Enddeposition()
LIN {X 0.6453,Y -92.375,Z 95,A -94.2999,B 24.9345,C -1.8698,E1 25.0007,E2 179.5092} C_DIS
Startdeposition()
$VEL.CP = VEL_PRINT
LIN {X -2.8024,Y -92.3395,Z 95,A -96.9309,B 24.9357,C -1.8527,E1 24.9932,E2 182.1811} C_DIS
LIN {X -6.5528,Y -92.1501,Z 95,A -99.3121,B 24.9357,C -1.8509,E1 24.9866,E2 184.5674} C_DIS
LIN {X -11.2683,Y -91.6939,Z 95,A -102.0824,B 24.9354,C -1.8569,E1 24.9789,E2 187.3252} C_DIS
LIN {X -15.8141,Y -91.0203,Z 95,A -104.9099,B 24.9353,C -1.8584,E1 24.9711,E2 190.1516} C_DIS
LIN {X -19.0565,Y -90.3967,Z 95,A -106.6609,B 24.9345,C -1.8691,E1 24.9664,E2 191.8792} C_DIS
LIN {X -21.5357,Y -89.8378,Z 95,A -108.4525,B 24.935,C -1.8628,E1 24.9615,E2 193.6883} C_DIS
LIN {X -24.0902,Y -89.186,Z 95,A -110.0308,B 24.9348,C -1.8656,E1 24.9572,E2 195.2621} C_DIS
LIN {X -27.4711,Y -88.2033,Z 95,A -112.2422,B 24.9348,C -1.8663,E1 24.9513,E2 197.4758} C_DIS
LIN {X -30.9192,Y -87.0552,Z 95,A -114.4271,B 24.9344,C -1.8704,E1 24.9455,E2 199.6551} C_DIS
LIN {X -33.6683,Y -86.0287,Z 95,A -116.3645,B 24.9346,C -1.8682,E1 24.9405,E2 201.6016} C_DIS
LIN {X -36.8349,Y -84.7212,Z 95,A -118.5797,B 24.9346,C -1.8675,E1 24.9348,E2 203.8237} C_DIS
LIN {X -40.3186,Y -83.1204,Z 95,A -120.7688,B 24.934,C -1.8764,E1 24.9293,E2 205.9973} C_DIS
LIN {X -43.3849,Y -81.5621,Z 95,A -123.1831,B 24.9344,C -1.8701,E1 24.9232,E2 208.4332} C_DIS
LIN {X -47.1962,Y -79.4169,Z 95,A -125.6672,B 24.9337,C -1.8812,E1 24.9173,E2 210.8982} C_DIS
LIN {X -54.0089,Y -74.9513,Z 95,A -130.8245,B 24.9333,C -1.8859,E1 24.9053,E2 216.0614} C_DIS
LIN {X -57.9857,Y -71.9179,Z 95,A -133.7643,B 24.9326,C -1.8966,E1 24.8988,E2 218.9864} C_DIS
LIN {X -60.2473,Y -70.0353,Z 95,A -135.7789,B 24.9327,C -1.8941,E1 24.8945,E2 221.0149} C_DIS
LIN {X -62.8819,Y -67.6804,Z 95,A -137.9126,B 24.9323,C -1.9002,E1 24.8901,E2 223.1424} C_DIS
LIN {X -65.1608,Y -65.4878,Z 95,A -139.8939,B 24.9321,C -1.9037,E1 24.8862,E2 225.1237} C_DIS
LIN {X -67.4991,Y -63.0748,Z 95,A -142.0337,B 24.9319,C -1.9065,E1 24.882,E2 227.2662} C_DIS
LIN {X -69.9285,Y -60.3718,Z 95,A -144.4008,B 24.9317,C -1.9081,E1 24.8777,E2 229.6403} C_DIS
LIN {X -72.6599,Y -57.0535,Z 95,A -147.6847,B 24.9327,C -1.8954,E1 24.8719,E2 232.9698} C_DIS
LIN {X -75.2282,Y -53.6209,Z 95,A -149.3696,B 24.93,C -1.9319,E1 24.8693,E2 234.5758} C_DIS
LIN {X -77.2282,Y -50.6983,Z 95,A -152.0049,B 24.9306,C -1.9239,E1 24.8651,E2 237.2433} C_DIS
LIN {X -79.6153,Y -46.8606,Z 95,A -154.6964,B 24.9298,C -1.9347,E1 24.8612,E2 239.923} C_DIS
LIN {X -81.2273,Y -44.0068,Z 95,A -156.8448,B 24.9297,C -1.9366,E1 24.8583,E2 242.0779} C_DIS
LIN {X -82.6482,Y -41.2775,Z 95,A -158.5472,B 24.9288,C -1.9482,E1 24.8562,E2 243.7619} C_DIS
LIN {X -83.9543,Y -38.5537,Z 95,A -160.5463,B 24.9288,C -1.9496,E1 24.8538,E2 245.7685} C_DIS
LIN {X -86.1674,Y -33.3144,Z 95,A -164.1778,B 24.9282,C -1.9566,E1 24.85,E2 249.4035} C_DIS
LIN {X -87.3406,Y -30.1057,Z 95,A -166.1983,B 24.9275,C -1.9659,E1 24.8481,E2 251.4135} C_DIS
LIN {X -88.3971,Y -26.8462,Z 95,A -168.4231,B 24.9273,C -1.9692,E1 24.8462,E2 253.6431} C_DIS
LIN {X -89.4439,Y -23.1144,Z 95,A -170.673,B 24.9264,C -1.9812,E1 24.8446,E2 255.8775} C_DIS
LIN {X -90.1778,Y -20.0645,Z 95,A -172.6371,B 24.926,C -1.9866,E1 24.8434,E2 257.8403} C_DIS
LIN {X -90.771,Y -17.1809,Z 95,A -174.8116,B 24.9264,C -1.9818,E1 24.8422,E2 260.039} C_DIS
LIN {X -91.3615,Y -13.7012,Z 95,A -176.7552,B 24.9253,C -1.996,E1 24.8414,E2 261.9603} C_DIS
LIN {X -91.7885,Y -10.4609,Z 95,A -178.976,B 24.9253,C -1.9966,E1 24.8406,E2 264.193} C_DIS
LIN {X -92.2075,Y -5.7045,Z 95,A 178.4256,B 24.9237,C -2.0169,E1 24.84,E2 266.7586} C_DIS
LIN {X -92.3293,Y -3.1409,Z 95,A 176.5942,B 24.9239,C -2.0148,E1 24.8398,E2 268.6061} C_DIS
LIN {X -92.3792,Y 0.8028,Z 95,A 174.0816,B 24.9234,C -2.0206,E1 24.8398,E2 271.1198} C_DIS
LIN {X -92.29,Y 4.13,Z 95,A 172.3693,B 24.9221,C -2.0378,E1 24.84,E2 272.8013} C_DIS
LIN {X -92.1518,Y 6.5281,Z 95,A 170.6216,B 24.9224,C -2.0348,E1 24.8403,E2 274.5667} C_DIS
LIN {X -91.8599,Y 9.8121,Z 95,A 168.5875,B 24.9218,C -2.0417,E1 24.8408,E2 276.5965} C_DIS
LIN {X -91.3712,Y 13.6385,Z 95,A 166.3461,B 24.9209,C -2.0539,E1 24.8417,E2 278.8222} C_DIS
LIN {X -90.641,Y 17.856,Z 95,A 163.4525,B 24.9208,C -2.0552,E1 24.8431,E2 281.7298} C_DIS
LIN {X -89.9109,Y 21.23,Z 95,A 161.3663,B 24.9201,C -2.0637,E1 24.8444,E2 283.8082} C_DIS
LIN {X -89.1325,Y 24.2882,Z 95,A 159.4146,B 24.9196,C -2.07,E1 24.8458,E2 285.7561} C_DIS
LIN {X -88.1129,Y 27.7629,Z 95,A 157.2327,B 24.9189,C -2.0789,E1 24.8475,E2 287.9293} C_DIS
LIN {X -87.1871,Y 30.5432,Z 95,A 154.888,B 24.9197,C -2.0688,E1 24.8497,E2 290.3116} C_DIS
LIN {X -85.8075,Y 34.2315,Z 95,A 152.7288,B 24.9185,C -2.0847,E1 24.8518,E2 292.4449} C_DIS
LIN {X -84.4198,Y 37.5234,Z 95,A 150.5635,B 24.9179,C -2.0929,E1 24.8542,E2 294.6026} C_DIS
LIN {X -82.9783,Y 40.6115,Z 95,A 148.372,B 24.9175,C -2.0969,E1 24.8569,E2 296.7966} C_DIS
LIN {X -81.3486,Y 43.7833,Z 95,A 145.7381,B 24.918,C -2.0907,E1 24.8604,E2 299.4591} C_DIS
LIN {X -79.7291,Y 46.6681,Z 95,A 144.3933,B 24.9159,C -2.1179,E1 24.8622,E2 300.7461} C_DIS
LIN {X -78.3169,Y 48.9994,Z 95,A 142.5443,B 24.9159,C -2.1179,E1 24.8649,E2 302.6046} C_DIS
LIN {X -76.5372,Y 51.7353,Z 95,A 140.4537,B 24.9156,C -2.1215,E1 24.8681,E2 304.697} C_DIS
LIN {X -74.9065,Y 54.0718,Z 95,A 138.6085,B 24.9154,C -2.1239,E1 24.8711,E2 306.5455} C_DIS
LIN {X -73.0513,Y 56.5511,Z 95,A 136.6734,B 24.915,C -2.1286,E1 24.8743,E2 308.4786} C_DIS
LIN {X -70.9346,Y 59.1844,Z 95,A 134.5093,B 24.9148,C -2.132,E1 24.8782,E2 310.6448} C_DIS
LIN {X -68.5886,Y 61.8887,Z 95,A 132.2979,B 24.9143,C -2.1379,E1 24.8823,E2 312.852} C_DIS
LIN {X -66.1934,Y 64.4446,Z 95,A 130.3219,B 24.9134,C -2.1492,E1 24.886,E2 314.8095} C_DIS
LIN {X -64.5332,Y 66.1078,Z 95,A 128.6336,B 24.9137,C -2.1456,E1 24.8894,E2 316.5136} C_DIS
LIN {X -62.1908,Y 68.3148,Z 95,A 126.6474,B 24.9133,C -2.1505,E1 24.8935,E2 318.496} C_DIS
LIN {X -59.5188,Y 70.6559,Z 95,A 124.359,B 24.9131,C -2.1528,E1 24.8983,E2 320.7878} C_DIS
LIN {X -57.2551,Y 72.5006,Z 95,A 122.7643,B 24.9122,C -2.1635,E1 24.9018,E2 322.3632} C_DIS
LIN {X -54.7848,Y 74.3853,Z 95,A 120.6688,B 24.9123,C -2.1622,E1 24.9065,E2 324.4691} C_DIS
LIN {X -51.6368,Y 76.6039,Z 95,A 118.2768,B 24.9119,C -2.1669,E1 24.912,E2 326.8582} C_DIS
LIN {X -48.5384,Y 78.6049,Z 95,A 116.0271,B 24.9115,C -2.1723,E1 24.9173,E2 329.1021} C_DIS
LIN {X -45.8035,Y 80.2283,Z 95,A 113.2489,B 24.9132,C -2.1508,E1 24.9242,E2 331.9398} C_DIS
LIN {X -41.8979,Y 82.3351,Z 95,A 111.3886,B 24.9106,C -2.1831,E1 24.9286,E2 333.7281} C_DIS
LIN {X -38.9935,Y 83.7495,Z 95,A 109.2393,B 24.9107,C -2.1817,E1 24.934,E2 335.8863} C_DIS
LIN {X -35.6312,Y 85.2348,Z 95,A 106.7948,B 24.9109,C -2.1798,E1 24.9403,E2 338.3412} C_DIS
LIN {X -31.8865,Y 86.7052,Z 95,A 104.5923,B 24.9098,C -2.1923,E1 24.946,E2 340.5183} C_DIS
LIN {X -28.8757,Y 87.7547,Z 95,A 102.4838,B 24.91,C -2.1906,E1 24.9516,E2 342.635} C_DIS
LIN {X -24.9868,Y 88.9392,Z 95,A 100.1057,B 24.9094,C -2.1979,E1 24.9579,E2 344.9996} C_DIS
LIN {X -22.152,Y 89.6874,Z 95,A 98.1364,B 24.9096,C -2.1949,E1 24.9633,E2 346.9791} C_DIS
LIN {X -18.775,Y 90.4545,Z 95,A 95.7014,B 24.9102,C -2.1875,E1 24.97,E2 349.4346} C_DIS
LIN {X -15.0449,Y 91.1491,Z 95,A 93.7702,B 24.909,C -2.2029,E1 24.9752,E2 351.3311} C_DIS
LIN {X -10.9292,Y 91.7337,Z 95,A 91.4256,B 24.9082,C -2.2121,E1 24.9816,E2 353.6556} C_DIS
LIN {X -8.5268,Y 91.9879,Z 95,A 89.6533,B 24.9089,C -2.2039,E1 24.9866,E2 355.4484} C_DIS
LIN {X -3.849,Y 92.3021,Z 95,A 86.693,B 24.9089,C -2.2033,E1 24.9949,E2 358.411} C_DIS
LIN {X 2.4382,Y 92.3509,Z 95,A 82.9093,B 24.9086,C -2.2079,E1 25.0054,E2 362.1838} C_DIS
LIN {X 5.9151,Y 92.1932,Z 95,A 80.528,B 24.9092,C -2.2005,E1 25.0121,E2 364.5817} C_DIS
LIN {X 10.0577,Y 91.8336,Z 95,A 77.6851,B 24.9099,C -2.1915,E1 25.02,E2 367.4442} C_DIS
LIN {X 15.7959,Y 91.0234,Z 95,A 74.5723,B 24.9087,C -2.2065,E1 25.0285,E2 370.5185} C_DIS
LIN {X 18.704,Y 90.4691,Z 95,A 72.5289,B 24.9093,C -2.1988,E1 25.0342,E2 372.5778} C_DIS
LIN {X 22.238,Y 89.6665,Z 95,A 70.2845,B 24.9094,C -2.1976,E1 25.0403,E2 374.8217} C_DIS
LIN {X 25.7054,Y 88.7356,Z 95,A 67.9578,B 24.9098,C -2.1927,E1 25.0465,E2 377.1562} C_DIS
LIN {X 29.5129,Y 87.5412,Z 95,A 65.6971,B 24.9094,C -2.198,E1 25.0525,E2 379.4001} C_DIS
LIN {X 32.5975,Y 86.4401,Z 95,A 63.6871,B 24.9094,C -2.1969,E1 25.0578,E2 381.4085} C_DIS
LIN {X 36.2944,Y 84.9553,Z 95,A 61.33,B 24.9094,C -2.1982,E1 25.0638,E2 383.7571} C_DIS
LIN {X 38.6279,Y 83.9197,Z 95,A 59.5017,B 24.9102,C -2.188,E1 25.0685,E2 385.605} C_DIS
LIN {X 42.1668,Y 82.1977,Z 95,A 57.0834,B 24.9104,C -2.1857,E1 25.0746,E2 388.0222} C_DIS
LIN {X 44.9554,Y 80.7062,Z 95,A 55.1445,B 24.9105,C -2.1838,E1 25.0793,E2 389.96} C_DIS
LIN {X 49.3457,Y 78.1006,Z 95,A 51.5962,B 24.912,C -2.1658,E1 25.0879,E2 393.5398} C_DIS
LIN {X 52.655,Y 75.9074,Z 95,A 49.6351,B 24.9109,C -2.1792,E1 25.0923,E2 395.4625} C_DIS
LIN {X 55.3081,Y 73.9969,Z 95,A 47.5486,B 24.9114,C -2.1737,E1 25.097,E2 397.5547} C_DIS
LIN {X 58.0973,Y 71.8275,Z 95,A 45.4249,B 24.9115,C -2.172,E1 25.1016,E2 399.6744} C_DIS
LIN {X 60.9832,Y 69.3946,Z 95,A 43.2069,B 24.9115,C -2.1719,E1 25.1063,E2 401.8842} C_DIS
LIN {X 63.0827,Y 67.4917,Z 95,A 41.2905,B 24.9123,C -2.1627,E1 25.1103,E2 403.8145} C_DIS
LIN {X 65.5809,Y 65.0666,Z 95,A 39.1337,B 24.9126,C -2.1582,E1 25.1146,E2 405.9728} C_DIS
LIN {X 68.3431,Y 62.16,Z 95,A 36.9006,B 24.9123,C -2.1618,E1 25.1188,E2 408.1878} C_DIS
LIN {X 71.0584,Y 59.0354,Z 95,A 34.2036,B 24.9132,C -2.1512,E1 25.1238,E2 410.8974} C_DIS
LIN {X 72.9283,Y 56.7107,Z 95,A 32.2415,B 24.9139,C -2.1428,E1 25.1272,E2 412.8703} C_DIS
LIN {X 75.1027,Y 53.7968,Z 95,A 30.0452,B 24.9142,C -2.1393,E1 25.1308,E2 415.0641} C_DIS
LIN {X 76.866,Y 51.2476,Z 95,A 28.1125,B 24.9146,C -2.1341,E1 25.1338,E2 416.9997} C_DIS
LIN {X 78.7091,Y 48.369,Z 95,A 26.0034,B 24.915,C -2.1289,E1 25.137,E2 419.1103} C_DIS
LIN {X 80.232,Y 45.7972,Z 95,A 23.2676,B 24.9179,C -2.0923,E1 25.1409,E2 421.9185} C_DIS
LIN {X 82.5325,Y 41.5109,Z 95,A 21.3384,B 24.9155,C -2.1231,E1 25.1432,E2 423.7647} C_DIS
LIN {X 84.7393,Y 36.7933,Z 95,A 17.9072,B 24.9168,C -2.1067,E1 25.1472,E2 427.2161} C_DIS
LIN {X 86.0515,Y 33.6102,Z 95,A 15.968,B 24.9167,C -2.1076,E1 25.1492,E2 429.1422} C_DIS
LIN {X 87.1396,Y 30.6786,Z 95,A 13.9156,B 24.9175,C -2.0978,E1 25.1512,E2 431.2064} C_DIS
LIN {X 88.1764,Y 27.5581,Z 95,A 11.9182,B 24.9178,C -2.0932,E1 25.1529,E2 433.2033} C_DIS
LIN {X 89.0575,Y 24.5659,Z 95,A 9.9966,B 24.9183,C -2.0878,E1 25.1544,E2 435.1267} C_DIS
LIN {X 90.3593,Y 19.2326,Z 95,A 6.7529,B 24.9186,C -2.0832,E1 25.1565,E2 438.3623} C_DIS
LIN {X 91.1245,Y 15.192,Z 95,A 4.2758,B 24.919,C -2.078,E1 25.1577,E2 440.8373} C_DIS
LIN {X 91.4912,Y 12.8017,Z 95,A 2.5343,B 24.9201,C -2.0644,E1 25.1584,E2 442.6007} C_DIS
LIN {X 91.8978,Y 9.45,Z 95,A 0.5114,B 24.9204,C -2.0604,E1 25.1591,E2 444.6211} C_DIS
LIN {X 92.1768,Y 6.1575,Z 95,A -1.5702,B 24.921,C -2.0526,E1 25.1595,E2 446.7086} C_DIS
LIN {X 92.3387,Y 2.8348,Z 95,A -3.5901,B 24.9214,C -2.0476,E1 25.1597,E2 448.7283} C_DIS
LIN {X 92.3464,Y -2.5859,Z 95,A -7.6074,B 24.924,C -2.0128,E1 25.1596,E2 452.8038} C_DIS
LIN {X 92.1488,Y -6.5692,Z 95,A -9.4464,B 24.9229,C -2.0281,E1 25.1593,E2 454.5959} C_DIS
LIN {X 91.2816,Y -14.2182,Z 95,A -13.613,B 24.9223,C -2.0352,E1 25.1579,E2 458.721} C_DIS
LIN {X 90.7088,Y -17.5042,Z 95,A -16.5369,B 24.9252,C -1.997,E1 25.1564,E2 461.7181} C_DIS
LIN {X 89.419,Y -23.2116,Z 95,A -19.588,B 24.9245,C -2.0068,E1 25.1545,E2 464.7284} C_DIS
LIN {X 88.7332,Y -25.7137,Z 95,A -21.4771,B 24.9256,C -1.9913,E1 25.153,E2 466.6431} C_DIS
LIN {X 87.6791,Y -29.104,Z 95,A -23.5732,B 24.9259,C -1.9884,E1 25.1513,E2 468.7344} C_DIS
LIN {X 86.6964,Y -31.9105,Z 95,A -25.4502,B 24.9264,C -1.9814,E1 25.1495,E2 470.6171} C_DIS
LIN {X 85.4769,Y -35.0462,Z 95,A -27.5423,B 24.9269,C -1.9748,E1 25.1473,E2 472.7132} C_DIS
LIN {X 83.9166,Y -38.6347,Z 95,A -29.9285,B 24.9273,C -1.969,E1 25.1446,E2 475.1002} C_DIS
LIN {X 82.6566,Y -41.2606,Z 95,A -31.5586,B 24.9273,C -1.9701,E1 25.1426,E2 476.719} C_DIS
LIN {X 81.2382,Y -43.9868,Z 95,A -33.616,B 24.9281,C -1.9589,E1 25.1399,E2 478.7919} C_DIS
LIN {X 79.7119,Y -46.6971,Z 95,A -35.5331,B 24.9284,C -1.9538,E1 25.1372,E2 480.7113} C_DIS
LIN {X 77.7294,Y -49.9261,Z 95,A -37.7047,B 24.9284,C -1.9536,E1 25.134,E2 482.8722} C_DIS
LIN {X 76.1142,Y -52.3575,Z 95,A -39.7081,B 24.9293,C -1.9415,E1 25.1309,E2 484.8943} C_DIS
LIN {X 73.9956,Y -55.3098,Z 95,A -42.0618,B 24.93,C -1.9317,E1 25.127,E2 487.2597} C_DIS
LIN {X 70.2816,Y -59.9581,Z 95,A -45.2749,B 24.9295,C -1.9394,E1 25.1214,E2 490.4398} C_DIS
LIN {X 68.7019,Y -61.7622,Z 95,A -47.025,B 24.9305,C -1.926,E1 25.1181,E2 492.2137} C_DIS
LIN {X 65.2204,Y -65.4284,Z 95,A -50.3054,B 24.9314,C -1.913,E1 25.1117,E2 495.5106} C_DIS
LIN {X 62.8873,Y -67.6754,Z 95,A -51.9983,B 24.9309,C -1.9197,E1 25.1083,E2 497.181} C_DIS
LIN {X 60.7727,Y -69.5784,Z 95,A -53.8478,B 24.9314,C -1.9126,E1 25.1044,E2 499.0399} C_DIS
LIN {X 57.515,Y -72.2952,Z 95,A -56.5046,B 24.9319,C -1.9058,E1 25.0987,E2 501.7026} C_DIS
LIN {X 55.3884,Y -73.9365,Z 95,A -58.2137,B 24.9323,C -1.9007,E1 25.0948,E2 503.4174} C_DIS
LIN {X 52.6753,Y -75.8933,Z 95,A -60.2626,B 24.9325,C -1.8974,E1 25.0902,E2 505.4671} C_DIS
LIN {X 49.6585,Y -77.9012,Z 95,A -62.5213,B 24.9328,C -1.8926,E1 25.0849,E2 507.7296} C_DIS
LIN {X 47.4203,Y -79.2844,Z 95,A -64.1125,B 24.933,C -1.891,E1 25.0811,E2 509.3197} C_DIS
LIN {X 45.038,Y -80.6602,Z 95,A -65.697,B 24.9329,C -1.8923,E1 25.0772,E2 510.8964} C_DIS
LIN {X 42.3117,Y -82.1236,Z 95,A -67.7044,B 24.9333,C -1.8859,E1 25.0723,E2 512.9133} C_DIS
LIN {X 39.5411,Y -83.494,Z 95,A -69.5072,B 24.9333,C -1.8869,E1 25.0677,E2 514.7091} C_DIS
LIN {X 36.7225,Y -84.7702,Z 95,A -71.5226,B 24.9337,C -1.8806,E1 25.0626,E2 516.7345} C_DIS
LIN {X 33.2841,Y -86.1795,Z 95,A -73.907,B 24.9341,C -1.8745,E1 25.0564,E2 519.1279} C_DIS
LIN {X 30.0195,Y -87.3704,Z 95,A -76.0653,B 24.9343,C -1.8716,E1 25.0507,E2 521.2886} C_DIS
LIN {X 26.6379,Y -88.4593,Z 95,A -78.3547,B 24.9347,C -1.866,E1 25.0446,E2 523.5871} C_DIS
LIN {X 21.4813,Y -89.8511,Z 95,A -81.898,B 24.9355,C -1.8547,E1 25.0349,E2 527.1518} C_DIS
LIN {X 16.8711,Y -90.8302,Z 95,A -85.462,B 24.9372,C -1.8304,E1 25.025,E2 530.7693} C_DIS
LIN {X 11.6584,Y -91.6439,Z 95,A -87.4944,B 24.9344,C -1.8705,E1 25.0196,E2 532.7049} C_DIS
LIN {X 6.5275,Y -92.1518,Z 95,A -90.8805,B 24.935,C -1.8624,E1 25.0102,E2 536.1083} C_DIS
LIN {X 4.2103,Y -92.2866,Z 95,A -92.707,B 24.9359,C -1.8487,E1 25.005,E2 537.9667} C_DIS
LIN {X 0.6453,Y -92.375,Z 95,A -94.2983,B 24.9345,C -1.8692,E1 25.0007,E2 539.5092} C_DIS
Enddeposition()
LIN {X 0.6453,Y -92.375,Z 95,A -94.2983,B 24.9345,C -1.8692,E1 25.0007,E2 539.5092} C_DIS
Startdeposition()
$VEL.CP = VEL_PRINT
LIN {X 1.5235,Y -91.4458,Z 95,A -93.2074,B 24.9321,C -1.9038,E1 25.004,E2 538.3364} C_DIS
LIN {X 4.1979,Y -91.3624,Z 95,A -91.4944,B 24.9319,C -1.9056,E1 25.0087,E2 536.6194} C_DIS
LIN {X 6.7047,Y -91.2138,Z 95,A -89.8074,B 24.9316,C -1.9102,E1 25.0135,E2 534.9223} C_DIS
LIN {X 9.2772,Y -90.9869,Z 95,A -88.1941,B 24.9316,C -1.911,E1 25.018,E2 533.3082} C_DIS
LIN {X 12.2895,Y -90.6305,Z 95,A -86.2931,B 24.9315,C -1.9122,E1 25.0232,E2 531.4059} C_DIS
LIN {X 15.211,Y -90.1847,Z 95,A -84.5248,B 24.9315,C -1.9107,E1 25.0281,E2 529.6429} C_DIS
LIN {X 18.1942,Y -89.6306,Z 95,A -82.7004,B 24.9316,C -1.9096,E1 25.0331,E2 527.8231} C_DIS
LIN {X 20.3684,Y -89.1617,Z 95,A -81.1948,B 24.9313,C -1.9148,E1 25.0372,E2 526.3072} C_DIS
LIN {X 23.594,Y -88.363,Z 95,A -79.1142,B 24.9311,C -1.9169,E1 25.0428,E2 524.2248} C_DIS
LIN {X 26.5475,Y -87.5224,Z 95,A -77.1497,B 24.9309,C -1.9205,E1 25.0481,E2 522.2553} C_DIS
LIN {X 29.3925,Y -86.6068,Z 95,A -75.388,B 24.9309,C -1.9189,E1 25.0528,E2 520.5006} C_DIS
LIN {X 32.1983,Y -85.6034,Z 95,A -73.5814,B 24.9309,C -1.9192,E1 25.0575,E2 518.697} C_DIS
LIN {X 34.4714,Y -84.7133,Z 95,A -71.921,B 24.9305,C -1.926,E1 25.0618,E2 517.0243} C_DIS
LIN {X 37.4119,Y -83.4566,Z 95,A -70.0602,B 24.9306,C -1.924,E1 25.0666,E2 515.1728} C_DIS
LIN {X 39.7861,Y -82.3513,Z 95,A -68.3708,B 24.9303,C -1.9283,E1 25.0708,E2 513.4776} C_DIS
LIN {X 42.1213,Y -81.1834,Z 95,A -66.6343,B 24.9298,C -1.9346,E1 25.0752,E2 511.731} C_DIS
LIN {X 44.4208,Y -79.9466,Z 95,A -65.0554,B 24.9298,C -1.9355,E1 25.079,E2 510.1547} C_DIS
LIN {X 47.0107,Y -78.4533,Z 95,A -63.1465,B 24.9294,C -1.9401,E1 25.0837,E2 508.2405} C_DIS
LIN {X 49.568,Y -76.8614,Z 95,A -61.3678,B 24.9294,C -1.9399,E1 25.0878,E2 506.4681} C_DIS
LIN {X 52.1144,Y -75.158,Z 95,A -59.543,B 24.9294,C -1.9403,E1 25.092,E2 504.6485} C_DIS
LIN {X 54.1722,Y -73.6888,Z 95,A -57.7199,B 24.9285,C -1.9522,E1 25.0962,E2 502.8037} C_DIS
LIN {X 56.8363,Y -71.6539,Z 95,A -55.6236,B 24.9282,C -1.9566,E1 25.1008,E2 500.7048} C_DIS
LIN {X 59.3126,Y -69.6179,Z 95,A -53.7368,B 24.9282,C -1.9567,E1 25.1048,E2 498.825} C_DIS
LIN {X 61.8228,Y -67.3986,Z 95,A -51.6456,B 24.9279,C -1.9613,E1 25.1092,E2 496.7314} C_DIS
LIN {X 64.2472,Y -65.0916,Z 95,A -49.5571,B 24.9275,C -1.966,E1 25.1134,E2 494.6404} C_DIS
LIN {X 66.6264,Y -62.6542,Z 95,A -47.4405,B 24.9272,C -1.9707,E1 25.1175,E2 492.5219} C_DIS
LIN {X 68.8769,Y -60.1714,Z 95,A -45.3503,B 24.9268,C -1.9757,E1 25.1214,E2 490.4292} C_DIS
LIN {X 71.0331,Y -57.6101,Z 95,A -43.2622,B 24.9264,C -1.9808,E1 25.1251,E2 488.3385} C_DIS
LIN {X 73.013,Y -55.0796,Z 95,A -41.3736,B 24.9264,C -1.9817,E1 25.1283,E2 486.4569} C_DIS
LIN {X 74.5581,Y -52.9693,Z 95,A -39.532,B 24.9255,C -1.9936,E1 25.1313,E2 484.5961} C_DIS
LIN {X 76.2426,Y -50.5148,Z 95,A -37.8914,B 24.9257,C -1.9906,E1 25.1339,E2 482.9708} C_DIS
LIN {X 77.4546,Y -48.636,Z 95,A -36.4996,B 24.9254,C -1.9942,E1 25.136,E2 481.5774} C_DIS
LIN {X 78.8309,Y -46.3718,Z 95,A -34.7953,B 24.925,C -2.0006,E1 25.1384,E2 479.8667} C_DIS
LIN {X 80.1239,Y -44.1033,Z 95,A -33.0637,B 24.9243,C -2.0089,E1 25.1408,E2 478.1246} C_DIS
LIN {X 81.3488,Y -41.7975,Z 95,A -31.5984,B 24.9244,C -2.0075,E1 25.1427,E2 476.6704} C_DIS
LIN {X 82.3481,Y -39.7927,Z 95,A -30.0589,B 24.9237,C -2.0167,E1 25.1446,E2 475.1174} C_DIS
LIN {X 83.7699,Y -36.705,Z 95,A -27.9821,B 24.9234,C -2.0212,E1 25.1469,E2 473.0413} C_DIS
LIN {X 84.9255,Y -33.9499,Z 95,A -26.23,B 24.9234,C -2.0224,E1 25.1488,E2 471.2958} C_DIS
LIN {X 85.8582,Y -31.5124,Z 95,A -24.6053,B 24.9229,C -2.0271,E1 25.1504,E2 469.6691} C_DIS
LIN {X 86.6041,Y -29.4007,Z 95,A -23.1023,B 24.9223,C -2.0352,E1 25.1518,E2 468.1555} C_DIS
LIN {X 87.5199,Y -26.5557,Z 95,A -21.1933,B 24.9218,C -2.0424,E1 25.1534,E2 466.2405} C_DIS
LIN {X 88.3393,Y -23.6819,Z 95,A -19.2692,B 24.9212,C -2.0502,E1 25.1548,E2 464.3089} C_DIS
LIN {X 89.1543,Y -20.4004,Z 95,A -17.3369,B 24.9212,C -2.0501,E1 25.156,E2 462.3881} C_DIS
LIN {X 89.7667,Y -17.5104,Z 95,A -15.4405,B 24.9206,C -2.0577,E1 25.1571,E2 460.4849} C_DIS
LIN {X 90.3161,Y -14.4163,Z 95,A -13.4958,B 24.9202,C -2.0631,E1 25.158,E2 458.5389} C_DIS
LIN {X 90.6693,Y -11.9903,Z 95,A -12.0833,B 24.9202,C -2.0634,E1 25.1585,E2 457.1338} C_DIS
LIN {X 91.0048,Y -9.1066,Z 95,A -10.0958,B 24.9192,C -2.0755,E1 25.1591,E2 455.1295} C_DIS
LIN {X 91.2348,Y -6.3949,Z 95,A -8.4654,B 24.919,C -2.0783,E1 25.1595,E2 453.5024} C_DIS
LIN {X 91.3927,Y -3.491,Z 95,A -6.5561,B 24.9183,C -2.0874,E1 25.1597,E2 451.5829} C_DIS
LIN {X 91.4584,Y -0.1895,Z 95,A -4.5462,B 24.9179,C -2.0918,E1 25.1597,E2 449.5744} C_DIS
LIN {X 91.4107,Y 2.956,Z 95,A -2.5249,B 24.9173,C -2.1,E1 25.1597,E2 447.5458} C_DIS
LIN {X 91.237,Y 6.3622,Z 95,A -0.4152,B 24.9168,C -2.1059,E1 25.1593,E2 445.4349} C_DIS
LIN {X 90.981,Y 9.3343,Z 95,A 1.3358,B 24.9168,C -2.1074,E1 25.1588,E2 443.6906} C_DIS
LIN {X 90.579,Y 12.6541,Z 95,A 3.3195,B 24.9165,C -2.1099,E1 25.1581,E2 441.7127} C_DIS
LIN {X 90.1693,Y 15.3028,Z 95,A 5.0299,B 24.916,C -2.1163,E1 25.1573,E2 439.9972} C_DIS
LIN {X 89.6273,Y 18.2102,Z 95,A 6.8116,B 24.9157,C -2.1195,E1 25.1564,E2 438.2185} C_DIS
LIN {X 89.1582,Y 20.3836,Z 95,A 8.3077,B 24.9151,C -2.1276,E1 25.1555,E2 436.7119} C_DIS
LIN {X 88.3424,Y 23.6702,Z 95,A 10.4146,B 24.9146,C -2.1335,E1 25.154,E2 434.6031} C_DIS
LIN {X 87.5242,Y 26.5416,Z 95,A 12.3216,B 24.9141,C -2.1405,E1 25.1525,E2 432.6906} C_DIS
LIN {X 86.61,Y 29.3831,Z 95,A 14.1904,B 24.9136,C -2.1461,E1 25.1508,E2 430.8192} C_DIS
LIN {X 85.5968,Y 32.2158,Z 95,A 15.8943,B 24.9137,C -2.145,E1 25.1492,E2 429.1274} C_DIS
LIN {X 84.7819,Y 34.3029,Z 95,A 17.2893,B 24.9134,C -2.1487,E1 25.1478,E2 427.7313} C_DIS
LIN {X 83.7648,Y 36.7167,Z 95,A 19.1391,B 24.9124,C -2.1611,E1 25.1457,E2 425.8624} C_DIS
LIN {X 82.3552,Y 39.778,Z 95,A 21.0718,B 24.9124,C -2.1605,E1 25.1434,E2 423.9416} C_DIS
LIN {X 81.1944,Y 42.0997,Z 95,A 22.7849,B 24.9118,C -2.1681,E1 25.1412,E2 422.2195} C_DIS
LIN {X 79.9687,Y 44.3812,Z 95,A 24.3609,B 24.9116,C -2.1709,E1 25.1391,E2 420.6453} C_DIS
LIN {X 78.4474,Y 47.0207,Z 95,A 26.1452,B 24.9116,C -2.1714,E1 25.1366,E2 418.8688} C_DIS
LIN {X 77.2721,Y 48.9281,Z 95,A 27.5413,B 24.9113,C -2.1748,E1 25.1345,E2 417.4718} C_DIS
LIN {X 76.0504,Y 50.8062,Z 95,A 28.9371,B 24.911,C -2.1781,E1 25.1324,E2 416.075} C_DIS
LIN {X 74.4318,Y 53.1463,Z 95,A 30.8115,B 24.9104,C -2.186,E1 25.1294,E2 414.1913} C_DIS
LIN {X 72.4433,Y 55.8265,Z 95,A 32.8966,B 24.91,C -2.1909,E1 25.1259,E2 412.1046} C_DIS
LIN {X 70.3442,Y 58.4494,Z 95,A 34.9939,B 24.9096,C -2.1956,E1 25.1222,E2 410.006} C_DIS
LIN {X 68.1428,Y 61.0015,Z 95,A 37.0989,B 24.9092,C -2.2001,E1 25.1183,E2 407.8996} C_DIS
LIN {X 65.8463,Y 63.4736,Z 95,A 39.1953,B 24.9089,C -2.2041,E1 25.1143,E2 405.8029} C_DIS
LIN {X 63.4711,Y 65.8487,Z 95,A 41.2906,B 24.9085,C -2.2083,E1 25.1101,E2 403.7067} C_DIS
LIN {X 61.0104,Y 68.1349,Z 95,A 43.3871,B 24.9082,C -2.2122,E1 25.1058,E2 401.6093} C_DIS
LIN {X 58.4537,Y 70.3406,Z 95,A 45.495,B 24.9079,C -2.216,E1 25.1013,E2 399.5006} C_DIS
LIN {X 55.8244,Y 72.4449,Z 95,A 47.5933,B 24.9076,C -2.2195,E1 25.0967,E2 397.4018} C_DIS
LIN {X 53.5823,Y 74.1207,Z 95,A 49.3989,B 24.9072,C -2.2243,E1 25.0926,E2 395.5913} C_DIS
LIN {X 51.4582,Y 75.609,Z 95,A 50.8315,B 24.9075,C -2.2203,E1 25.0893,E2 394.1731} C_DIS
LIN {X 49.0801,Y 77.1746,Z 95,A 52.6375,B 24.9072,C -2.2239,E1 25.0851,E2 392.3645} C_DIS
LIN {X 47.279,Y 78.2904,Z 95,A 54.1515,B 24.9065,C -2.2324,E1 25.0814,E2 390.835} C_DIS
LIN {X 44.4286,Y 79.9422,Z 95,A 56.223,B 24.9062,C -2.2356,E1 25.0764,E2 388.7622} C_DIS
LIN {X 41.7987,Y 81.3482,Z 95,A 57.9639,B 24.9064,C -2.2336,E1 25.0721,E2 387.0308} C_DIS
LIN {X 39.1027,Y 82.6796,Z 95,A 59.8409,B 24.9062,C -2.2356,E1 25.0674,E2 385.1539} C_DIS
LIN {X 36.7317,Y 83.7583,Z 95,A 61.489,B 24.906,C -2.238,E1 25.0632,E2 383.5042} C_DIS
LIN {X 33.7391,Y 85.0083,Z 95,A 63.5669,B 24.9057,C -2.2417,E1 25.0578,E2 381.4224} C_DIS
LIN {X 30.465,Y 86.2354,Z 95,A 65.5922,B 24.906,C -2.238,E1 25.0525,E2 379.41} C_DIS
LIN {X 27.9824,Y 87.0727,Z 95,A 67.2929,B 24.9058,C -2.2414,E1 25.048,E2 377.7045} C_DIS
LIN {X 25.1136,Y 87.943,Z 95,A 69.215,B 24.9055,C -2.2443,E1 25.0428,E2 375.779} C_DIS
LIN {X 21.8673,Y 88.8059,Z 95,A 71.3178,B 24.9055,C -2.2455,E1 25.0372,E2 373.6765} C_DIS
LIN {X 18.941,Y 89.4773,Z 95,A 73.2464,B 24.9052,C -2.248,E1 25.0319,E2 371.7444} C_DIS
LIN {X 16.0122,Y 90.0459,Z 95,A 75.0085,B 24.9054,C -2.2452,E1 25.0271,E2 369.9911} C_DIS
LIN {X 13.0499,Y 90.5227,Z 95,A 76.8278,B 24.9056,C -2.2437,E1 25.0221,E2 368.177} C_DIS
LIN {X 10.8486,Y 90.8129,Z 95,A 78.3324,B 24.9052,C -2.2478,E1 25.0179,E2 366.6638} C_DIS
LIN {X 7.5457,Y 91.1469,Z 95,A 80.2921,B 24.9055,C -2.244,E1 25.0125,E2 364.7143} C_DIS
LIN {X 4.619,Y 91.3426,Z 95,A 82.3238,B 24.905,C -2.2504,E1 25.0068,E2 362.6681} C_DIS
LIN {X 1.5062,Y 91.4461,Z 95,A 84.1451,B 24.9054,C -2.2459,E1 25.0017,E2 360.8579} C_DIS
LIN {X -1.4454,Y 91.4472,Z 95,A 85.9343,B 24.9056,C -2.2435,E1 24.9967,E2 359.0744} C_DIS
Enddeposition()
END
